ABB RAPID module: 01400AE1

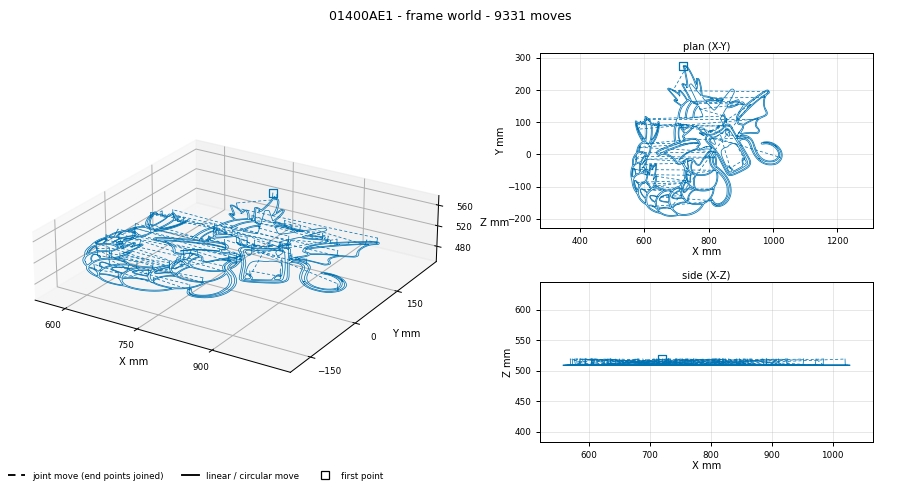
[picture p0: tool path of 01400AE1 in frame world, 9331 of 9331 moves have a stored position in this frame; points joined in program order, loops and branches not executed]
MODULE Module1
    !***********************************************************
    !
    ! Module:  Module1
    !
    ! Description:
    !   <Insert description here>
    !
    ! Author: ufabc
    !
    ! Version: 1.0
    !
    !***********************************************************


    !***********************************************************
    !
    ! Procedure main
    !
    !   This is the entry point of your program
    !
    !***********************************************************
    PROC main()
        !Add your code here
        CONST robtarget p0:=[[557.96,-192.62,509.20],[0.00299687,-0.165444,-0.986215,-0.000502744],[-1,0,0,0],[9E+09,9E+09,9E+09,9E+09,9E+09,9E+09]];

      MoveJ Offs(p0,163.0,466.8, 10), v100, z1, tool0;
MoveL Offs(p0,163.22140000000005,465.1791, 0), v100, z5, tool0;
MoveL Offs(p0,163.3808,464.47520000000003, 0), v100, z5, tool0;
MoveL Offs(p0,163.575,463.7125, 0), v100, z5, tool0;
MoveL Offs(p0,163.79919999999998,462.90479999999997, 0), v100, z5, tool0;
MoveL Offs(p0,164.0486,462.06589999999994, 0), v100, z5, tool0;
MoveL Offs(p0,164.31840000000003,461.2096, 0), v100, z5, tool0;
MoveL Offs(p0,164.6038,460.34970000000004, 0), v100, z5, tool0;
MoveL Offs(p0,164.9,459.5, 0), v100, z5, tool0;
MoveL Offs(p0,165.8568,456.4537, 0), v100, z5, tool0;
MoveL Offs(p0,166.95040000000003,452.1936000000002, 0), v100, z5, tool0;
MoveL Offs(p0,168.12560000000002,447.01789999999994, 0), v100, z5, tool0;
MoveL Offs(p0,169.3272,441.2248000000001, 0), v100, z5, tool0;
MoveL Offs(p0,170.5,435.1125, 0), v100, z5, tool0;
MoveL Offs(p0,171.5888,428.97919999999993, 0), v100, z5, tool0;
MoveL Offs(p0,172.5384,423.12309999999997, 0), v100, z5, tool0;
MoveL Offs(p0,173.29360000000003,417.8424000000001, 0), v100, z5, tool0;
MoveL Offs(p0,173.7992,413.4353, 0), v100, z5, tool0;
MoveL Offs(p0,174.0,410.2, 0), v100, z5, tool0;
MoveL Offs(p0,174.0,407.8, 0), v100, z5, tool0;
MoveL Offs(p0,169.4,410.4, 0), v100, z5, tool0;
MoveL Offs(p0,167.8938,411.19489999999996, 0), v100, z5, tool0;
MoveL Offs(p0,166.49440000000007,411.83920000000006, 0), v100, z5, tool0;
MoveL Offs(p0,165.20059999999998,412.33230000000003, 0), v100, z5, tool0;
MoveL Offs(p0,164.0112,412.67359999999996, 0), v100, z5, tool0;
MoveL Offs(p0,162.925,412.8625, 0), v100, z5, tool0;
MoveL Offs(p0,161.9408,412.8983999999999, 0), v100, z5, tool0;
MoveL Offs(p0,161.05739999999997,412.78069999999997, 0), v100, z5, tool0;
MoveL Offs(p0,160.27360000000002,412.50880000000006, 0), v100, z5, tool0;
MoveL Offs(p0,159.5882,412.08209999999997, 0), v100, z5, tool0;
MoveL Offs(p0,159.0,411.5, 0), v100, z5, tool0;
MoveL Offs(p0,158.76520000000002,411.12570000000005, 0), v100, z5, tool0;
MoveL Offs(p0,158.66960000000003,410.6416000000001, 0), v100, z5, tool0;
MoveL Offs(p0,158.72639999999998,410.01590000000004, 0), v100, z5, tool0;
MoveL Offs(p0,159.35,408.2125, 0), v100, z5, tool0;
MoveL Offs(p0,159.9432,406.9712, 0), v100, z5, tool0;
MoveL Offs(p0,160.7416,405.4611, 0), v100, z5, tool0;
MoveL Offs(p0,161.75840000000002,403.65040000000005, 0), v100, z5, tool0;
MoveL Offs(p0,163.00680000000003,401.50730000000004, 0), v100, z5, tool0;
MoveL Offs(p0,164.5,399.0, 0), v100, z5, tool0;
MoveL Offs(p0,166.88540000000003,394.95990000000006, 0), v100, z5, tool0;
MoveL Offs(p0,169.31520000000003,390.7272000000001, 0), v100, z5, tool0;
MoveL Offs(p0,171.71980000000002,386.43330000000003, 0), v100, z5, tool0;
MoveL Offs(p0,174.02960000000002,382.2096, 0), v100, z5, tool0;
MoveL Offs(p0,176.175,378.1875, 0), v100, z5, tool0;
MoveL Offs(p0,178.08639999999997,374.49839999999995, 0), v100, z5, tool0;
MoveL Offs(p0,179.6942,371.2737, 0), v100, z5, tool0;
MoveL Offs(p0,180.9288,368.64480000000003, 0), v100, z5, tool0;
MoveL Offs(p0,181.72060000000002,366.7431, 0), v100, z5, tool0;
MoveL Offs(p0,182.0,365.7, 0), v100, z5, tool0;
MoveL Offs(p0,181.59200000000004,364.89280000000014, 0), v100, z5, tool0;
MoveL Offs(p0,181.136,364.41569999999996, 0), v100, z5, tool0;
MoveL Offs(p0,180.56,363.92240000000004, 0), v100, z5, tool0;
MoveL Offs(p0,179.9,363.4375, 0), v100, z5, tool0;
MoveL Offs(p0,179.19199999999998,362.98560000000003, 0), v100, z5, tool0;
MoveL Offs(p0,178.47199999999998,362.5913, 0), v100, z5, tool0;
MoveL Offs(p0,177.776,362.27920000000006, 0), v100, z5, tool0;
MoveL Offs(p0,177.14000000000001,362.07390000000004, 0), v100, z5, tool0;
MoveL Offs(p0,176.6,362.0, 0), v100, z5, tool0;
MoveL Offs(p0,176.25680000000006,362.4672000000001, 0), v100, z5, tool0;
MoveL Offs(p0,175.8917,363.0233, 0), v100, z5, tool0;
MoveL Offs(p0,175.41440000000003,363.7696000000001, 0), v100, z5, tool0;
MoveL Offs(p0,174.8375,364.6875, 0), v100, z5, tool0;
MoveL Offs(p0,174.17360000000002,365.7584, 0), v100, z5, tool0;
MoveL Offs(p0,173.43529999999998,366.96369999999996, 0), v100, z5, tool0;
MoveL Offs(p0,172.63520000000003,368.2848, 0), v100, z5, tool0;
MoveL Offs(p0,171.7859,369.7031, 0), v100, z5, tool0;
MoveL Offs(p0,170.9,371.2, 0), v100, z5, tool0;
MoveL Offs(p0,169.93810000000002,372.75730000000004, 0), v100, z5, tool0;
MoveL Offs(p0,168.86880000000002,374.40640000000013, 0), v100, z5, tool0;
MoveL Offs(p0,167.7167,376.1131, 0), v100, z5, tool0;
MoveL Offs(p0,166.5064,377.8432, 0), v100, z5, tool0;
MoveL Offs(p0,165.2625,379.5625, 0), v100, z5, tool0;
MoveL Offs(p0,164.0096,381.23679999999996, 0), v100, z5, tool0;
MoveL Offs(p0,162.7723,382.8319, 0), v100, z5, tool0;
MoveL Offs(p0,161.57520000000002,384.31360000000006, 0), v100, z5, tool0;
MoveL Offs(p0,160.4429,385.64770000000004, 0), v100, z5, tool0;
MoveL Offs(p0,159.4,386.8, 0), v100, z5, tool0;
MoveL Offs(p0,157.8607,388.40900000000005, 0), v100, z5, tool0;
MoveL Offs(p0,156.57760000000002,389.7120000000001, 0), v100, z5, tool0;
MoveL Offs(p0,155.5129,390.733, 0), v100, z5, tool0;
MoveL Offs(p0,154.6288,391.49600000000004, 0), v100, z5, tool0;
MoveL Offs(p0,153.8875,392.025, 0), v100, z5, tool0;
MoveL Offs(p0,153.25119999999998,392.34399999999994, 0), v100, z5, tool0;
MoveL Offs(p0,152.6821,392.477, 0), v100, z5, tool0;
MoveL Offs(p0,152.1424,392.44800000000004, 0), v100, z5, tool0;
MoveL Offs(p0,151.59430000000003,392.281, 0), v100, z5, tool0;
MoveL Offs(p0,151.0,392.0, 0), v100, z5, tool0;
MoveL Offs(p0,150.4772,391.7028, 0), v100, z5, tool0;
MoveL Offs(p0,150.04560000000004,391.3984000000001, 0), v100, z5, tool0;
MoveL Offs(p0,149.70039999999997,391.06759999999997, 0), v100, z5, tool0;
MoveL Offs(p0,149.4368,390.69120000000004, 0), v100, z5, tool0;
MoveL Offs(p0,149.25,390.25, 0), v100, z5, tool0;
MoveL Offs(p0,149.13520000000003,389.7248, 0), v100, z5, tool0;
MoveL Offs(p0,149.0876,389.0964, 0), v100, z5, tool0;
MoveL Offs(p0,149.10240000000002,388.3456, 0), v100, z5, tool0;
MoveL Offs(p0,149.1748,387.45320000000004, 0), v100, z5, tool0;
MoveL Offs(p0,149.3,386.4, 0), v100, z5, tool0;
MoveL Offs(p0,149.51680000000005,384.25440000000015, 0), v100, z5, tool0;
MoveL Offs(p0,149.5502,383.5281, 0), v100, z5, tool0;
MoveL Offs(p0,149.5224,383.01120000000003, 0), v100, z5, tool0;
MoveL Offs(p0,148.98780000000002,382.5549, 0), v100, z5, tool0;
MoveL Offs(p0,148.6312,382.71360000000004, 0), v100, z5, tool0;
MoveL Offs(p0,148.1714,383.0007, 0), v100, z5, tool0;
MoveL Offs(p0,147.6,383.4, 0), v100, z5, tool0;
MoveL Offs(p0,145.2276,385.0427000000001, 0), v100, z5, tool0;
MoveL Offs(p0,142.50480000000005,386.80960000000016, 0), v100, z5, tool0;
MoveL Offs(p0,139.5432,388.6389, 0), v100, z5, tool0;
MoveL Offs(p0,136.45440000000002,390.46880000000004, 0), v100, z5, tool0;
MoveL Offs(p0,133.35,392.2375, 0), v100, z5, tool0;
MoveL Offs(p0,130.3416,393.88319999999993, 0), v100, z5, tool0;
MoveL Offs(p0,127.54079999999999,395.34409999999997, 0), v100, z5, tool0;
MoveL Offs(p0,125.0592,396.5584, 0), v100, z5, tool0;
MoveL Offs(p0,123.00840000000001,397.4643, 0), v100, z5, tool0;
MoveL Offs(p0,121.5,398.0, 0), v100, z5, tool0;
MoveL Offs(p0,120.39220000000003,398.29670000000004, 0), v100, z5, tool0;
MoveL Offs(p0,119.45360000000002,398.52560000000005, 0), v100, z5, tool0;
MoveL Offs(p0,118.6614,398.6848999999999, 0), v100, z5, tool0;
MoveL Offs(p0,117.99279999999999,398.7728000000001, 0), v100, z5, tool0;
MoveL Offs(p0,117.425,398.7875, 0), v100, z5, tool0;
MoveL Offs(p0,116.93519999999998,398.7272, 0), v100, z5, tool0;
MoveL Offs(p0,116.5006,398.5901, 0), v100, z5, tool0;
MoveL Offs(p0,116.0984,398.37440000000004, 0), v100, z5, tool0;
MoveL Offs(p0,115.3,397.7, 0), v100, z5, tool0;
MoveL Offs(p0,114.80490000000002,397.22830000000005, 0), v100, z5, tool0;
MoveL Offs(p0,114.47120000000004,396.7944000000001, 0), v100, z5, tool0;
MoveL Offs(p0,114.40630000000002,396.2501, 0), v100, z5, tool0;
MoveL Offs(p0,114.71759999999999,395.4472, 0), v100, z5, tool0;
MoveL Offs(p0,115.5125,394.2375, 0), v100, z5, tool0;
MoveL Offs(p0,116.89840000000001,392.4728, 0), v100, z5, tool0;
MoveL Offs(p0,118.9827,390.0049, 0), v100, z5, tool0;
MoveL Offs(p0,121.87280000000001,386.6856000000001, 0), v100, z5, tool0;
MoveL Offs(p0,125.67609999999999,382.36670000000004, 0), v100, z5, tool0;
MoveL Offs(p0,130.5,376.9, 0), v100, z5, tool0;
MoveL Offs(p0,141.4,364.5, 0), v100, z5, tool0;
MoveL Offs(p0,138.0,364.0, 0), v100, z5, tool0;
MoveL Offs(p0,136.66540000000003,363.7148, 0), v100, z5, tool0;
MoveL Offs(p0,135.60320000000004,363.2904000000001, 0), v100, z5, tool0;
MoveL Offs(p0,134.81580000000002,362.74359999999996, 0), v100, z5, tool0;
MoveL Offs(p0,134.3056,362.0912, 0), v100, z5, tool0;
MoveL Offs(p0,134.075,361.35, 0), v100, z5, tool0;
MoveL Offs(p0,134.1264,360.53679999999997, 0), v100, z5, tool0;
MoveL Offs(p0,134.4622,359.6684, 0), v100, z5, tool0;
MoveL Offs(p0,135.0848,358.76160000000004, 0), v100, z5, tool0;
MoveL Offs(p0,135.9966,357.83320000000003, 0), v100, z5, tool0;
MoveL Offs(p0,137.2,356.9, 0), v100, z5, tool0;
MoveL Offs(p0,137.83499999999998,356.468, 0), v100, z5, tool0;
MoveL Offs(p0,138.64400000000006,355.9040000000001, 0), v100, z5, tool0;
MoveL Offs(p0,139.603,355.226, 0), v100, z5, tool0;
MoveL Offs(p0,140.68800000000002,354.45200000000006, 0), v100, z5, tool0;
MoveL Offs(p0,141.875,353.6, 0), v100, z5, tool0;
MoveL Offs(p0,143.14000000000001,352.688, 0), v100, z5, tool0;
MoveL Offs(p0,144.459,351.73400000000004, 0), v100, z5, tool0;
MoveL Offs(p0,145.80800000000002,350.75600000000003, 0), v100, z5, tool0;
MoveL Offs(p0,147.163,349.77200000000005, 0), v100, z5, tool0;
MoveL Offs(p0,148.5,348.8, 0), v100, z5, tool0;
MoveL Offs(p0,156.6,342.9, 0), v100, z5, tool0;
MoveL Offs(p0,153.3,336.2, 0), v100, z5, tool0;
MoveL Offs(p0,152.22450000000003,333.89, 0), v100, z5, tool0;
MoveL Offs(p0,151.22400000000005,331.4240000000001, 0), v100, z5, tool0;
MoveL Offs(p0,150.30749999999998,328.838, 0), v100, z5, tool0;
MoveL Offs(p0,149.48399999999998,326.168, 0), v100, z5, tool0;
MoveL Offs(p0,148.7625,323.45, 0), v100, z5, tool0;
MoveL Offs(p0,148.152,320.72, 0), v100, z5, tool0;
MoveL Offs(p0,147.6615,318.014, 0), v100, z5, tool0;
MoveL Offs(p0,147.3,315.36800000000005, 0), v100, z5, tool0;
MoveL Offs(p0,147.07649999999998,312.81800000000004, 0), v100, z5, tool0;
MoveL Offs(p0,147.0,310.4, 0), v100, z5, tool0;
MoveL Offs(p0,146.7536,306.6048, 0), v100, z5, tool0;
MoveL Offs(p0,146.575,306.025, 0), v100, z5, tool0;
MoveL Offs(p0,146.3304,305.5472, 0), v100, z5, tool0;
MoveL Offs(p0,146.0102,305.1486, 0), v100, z5, tool0;
MoveL Offs(p0,145.6048,304.80640000000005, 0), v100, z5, tool0;
MoveL Offs(p0,145.1046,304.4978, 0), v100, z5, tool0;
MoveL Offs(p0,144.5,304.2, 0), v100, z5, tool0;
MoveL Offs(p0,143.69200000000004,303.78720000000004, 0), v100, z5, tool0;
MoveL Offs(p0,143.321,303.54929999999996, 0), v100, z5, tool0;
MoveL Offs(p0,142.98000000000002,303.2976, 0), v100, z5, tool0;
MoveL Offs(p0,142.675,303.0375, 0), v100, z5, tool0;
MoveL Offs(p0,142.412,302.7744, 0), v100, z5, tool0;
MoveL Offs(p0,142.197,302.5137, 0), v100, z5, tool0;
MoveL Offs(p0,142.036,302.2608, 0), v100, z5, tool0;
MoveL Offs(p0,141.935,302.02110000000005, 0), v100, z5, tool0;
MoveL Offs(p0,141.9,301.8, 0), v100, z5, tool0;
MoveL Offs(p0,141.7,299.85, 0), v100, z5, tool0;
MoveL Offs(p0,141.65519999999998,299.3088, 0), v100, z5, tool0;
MoveL Offs(p0,141.6116,298.7424, 0), v100, z5, tool0;
MoveL Offs(p0,141.5704,298.1616, 0), v100, z5, tool0;
MoveL Offs(p0,141.5328,297.5772, 0), v100, z5, tool0;
MoveL Offs(p0,141.5,297.0, 0), v100, z5, tool0;
MoveL Offs(p0,141.22160000000002,295.45040000000006, 0), v100, z5, tool0;
MoveL Offs(p0,140.9744,294.4071, 0), v100, z5, tool0;
MoveL Offs(p0,140.6648,293.2192, 0), v100, z5, tool0;
MoveL Offs(p0,140.3,291.9125, 0), v100, z5, tool0;
MoveL Offs(p0,139.88719999999998,290.51279999999997, 0), v100, z5, tool0;
MoveL Offs(p0,139.4336,289.04589999999996, 0), v100, z5, tool0;
MoveL Offs(p0,138.94639999999998,287.5376, 0), v100, z5, tool0;
MoveL Offs(p0,138.4328,286.0137, 0), v100, z5, tool0;
MoveL Offs(p0,137.9,284.5, 0), v100, z5, tool0;
MoveL Offs(p0,137.07820000000004,282.18640000000005, 0), v100, z5, tool0;
MoveL Offs(p0,136.40160000000006,280.1512000000001, 0), v100, z5, tool0;
MoveL Offs(p0,135.8534,278.28279999999995, 0), v100, z5, tool0;
MoveL Offs(p0,135.41680000000002,276.4696, 0), v100, z5, tool0;
MoveL Offs(p0,135.075,274.6, 0), v100, z5, tool0;
MoveL Offs(p0,134.81119999999999,272.56239999999997, 0), v100, z5, tool0;
MoveL Offs(p0,134.6086,270.2452, 0), v100, z5, tool0;
MoveL Offs(p0,134.4504,267.53679999999997, 0), v100, z5, tool0;
MoveL Offs(p0,134.31980000000001,264.3256, 0), v100, z5, tool0;
MoveL Offs(p0,134.2,260.5, 0), v100, z5, tool0;
MoveL Offs(p0,134.6125,243.425, 0), v100, z5, tool0;
MoveL Offs(p0,134.97039999999998,240.6424, 0), v100, z5, tool0;
MoveL Offs(p0,135.4327,237.92219999999998, 0), v100, z5, tool0;
MoveL Offs(p0,136.00480000000002,235.2008, 0), v100, z5, tool0;
MoveL Offs(p0,136.6921,232.4146, 0), v100, z5, tool0;
MoveL Offs(p0,137.5,229.5, 0), v100, z5, tool0;
MoveL Offs(p0,137.15169999999998,227.925, 0), v100, z5, tool0;
MoveL Offs(p0,136.46640000000002,227.36399999999998, 0), v100, z5, tool0;
MoveL Offs(p0,135.3875,226.725, 0), v100, z5, tool0;
MoveL Offs(p0,133.8496,225.97200000000004, 0), v100, z5, tool0;
MoveL Offs(p0,131.78730000000002,225.06900000000002, 0), v100, z5, tool0;
MoveL Offs(p0,129.1352,223.98000000000002, 0), v100, z5, tool0;
MoveL Offs(p0,125.8279,222.669, 0), v100, z5, tool0;
MoveL Offs(p0,121.8,221.1, 0), v100, z5, tool0;
MoveL Offs(p0,115.05690000000001,218.44700000000003, 0), v100, z5, tool0;
MoveL Offs(p0,108.97920000000002,216.00400000000008, 0), v100, z5, tool0;
MoveL Offs(p0,103.55429999999998,213.76500000000001, 0), v100, z5, tool0;
MoveL Offs(p0,98.7696,211.72400000000002, 0), v100, z5, tool0;
MoveL Offs(p0,94.6125,209.875, 0), v100, z5, tool0;
MoveL Offs(p0,91.07039999999999,208.212, 0), v100, z5, tool0;
MoveL Offs(p0,88.1307,206.72899999999998, 0), v100, z5, tool0;
MoveL Offs(p0,85.7808,205.42, 0), v100, z5, tool0;
MoveL Offs(p0,84.0081,204.279, 0), v100, z5, tool0;
MoveL Offs(p0,82.8,203.3, 0), v100, z5, tool0;
MoveL Offs(p0,81.75000000000001,202.14080000000004, 0), v100, z5, tool0;
MoveL Offs(p0,80.94000000000003,200.95040000000006, 0), v100, z5, tool0;
MoveL Offs(p0,80.37,199.73959999999997, 0), v100, z5, tool0;
MoveL Offs(p0,80.04,198.5192, 0), v100, z5, tool0;
MoveL Offs(p0,79.95,197.3, 0), v100, z5, tool0;
MoveL Offs(p0,80.1,196.09279999999998, 0), v100, z5, tool0;
MoveL Offs(p0,80.49000000000001,194.90839999999997, 0), v100, z5, tool0;
MoveL Offs(p0,81.12,193.7576, 0), v100, z5, tool0;
MoveL Offs(p0,81.99000000000001,192.65120000000002, 0), v100, z5, tool0;
MoveL Offs(p0,83.1,191.6, 0), v100, z5, tool0;
MoveL Offs(p0,84.1761,190.75700000000003, 0), v100, z5, tool0;
MoveL Offs(p0,85.19280000000003,190.08800000000002, 0), v100, z5, tool0;
MoveL Offs(p0,86.1627,189.59300000000002, 0), v100, z5, tool0;
MoveL Offs(p0,87.0984,189.272, 0), v100, z5, tool0;
MoveL Offs(p0,88.0125,189.125, 0), v100, z5, tool0;
MoveL Offs(p0,88.91760000000001,189.152, 0), v100, z5, tool0;
MoveL Offs(p0,89.82629999999999,189.353, 0), v100, z5, tool0;
MoveL Offs(p0,90.75120000000001,189.728, 0), v100, z5, tool0;
MoveL Offs(p0,91.70490000000001,190.277, 0), v100, z5, tool0;
MoveL Offs(p0,92.7,191.0, 0), v100, z5, tool0;
MoveL Offs(p0,94.55320000000002,192.03410000000002, 0), v100, z5, tool0;
MoveL Offs(p0,96.88160000000002,192.68480000000002, 0), v100, z5, tool0;
MoveL Offs(p0,99.60839999999999,192.9647, 0), v100, z5, tool0;
MoveL Offs(p0,102.65680000000002,192.88640000000004, 0), v100, z5, tool0;
MoveL Offs(p0,105.95,192.4625, 0), v100, z5, tool0;
MoveL Offs(p0,109.41120000000001,191.7056, 0), v100, z5, tool0;
MoveL Offs(p0,112.9636,190.6283, 0), v100, z5, tool0;
MoveL Offs(p0,116.53040000000001,189.24320000000003, 0), v100, z5, tool0;
MoveL Offs(p0,120.03479999999999,187.56289999999998, 0), v100, z5, tool0;
MoveL Offs(p0,123.4,185.6, 0), v100, z5, tool0;
MoveL Offs(p0,125.15720000000002,184.40070000000003, 0), v100, z5, tool0;
MoveL Offs(p0,126.88560000000003,183.08560000000006, 0), v100, z5, tool0;
MoveL Offs(p0,128.5804,181.65890000000002, 0), v100, z5, tool0;
MoveL Offs(p0,130.23680000000002,180.1248, 0), v100, z5, tool0;
MoveL Offs(p0,131.85,178.4875, 0), v100, z5, tool0;
MoveL Offs(p0,133.4152,176.75119999999998, 0), v100, z5, tool0;
MoveL Offs(p0,134.92759999999998,174.9201, 0), v100, z5, tool0;
MoveL Offs(p0,136.38240000000002,172.9984, 0), v100, z5, tool0;
MoveL Offs(p0,137.7748,170.99030000000002, 0), v100, z5, tool0;
MoveL Offs(p0,139.1,168.9, 0), v100, z5, tool0;
MoveL Offs(p0,140.6022,166.75030000000004, 0), v100, z5, tool0;
MoveL Offs(p0,142.2136,164.92640000000003, 0), v100, z5, tool0;
MoveL Offs(p0,143.91140000000001,163.4361, 0), v100, z5, tool0;
MoveL Offs(p0,145.6728,162.2872, 0), v100, z5, tool0;
MoveL Offs(p0,147.475,161.4875, 0), v100, z5, tool0;
MoveL Offs(p0,149.2952,161.04479999999998, 0), v100, z5, tool0;
MoveL Offs(p0,151.1106,160.96689999999998, 0), v100, z5, tool0;
MoveL Offs(p0,152.8984,161.2616, 0), v100, z5, tool0;
MoveL Offs(p0,154.63580000000002,161.93670000000003, 0), v100, z5, tool0;
MoveL Offs(p0,156.3,163.0, 0), v100, z5, tool0;
MoveL Offs(p0,158.9,165.1, 0), v100, z5, tool0;
MoveL Offs(p0,161.4,160.3, 0), v100, z5, tool0;
MoveL Offs(p0,161.84230000000002,159.48710000000003, 0), v100, z5, tool0;
MoveL Offs(p0,162.32240000000007,158.6208000000001, 0), v100, z5, tool0;
MoveL Offs(p0,162.83009999999996,157.7197, 0), v100, z5, tool0;
MoveL Offs(p0,163.35520000000002,156.8024, 0), v100, z5, tool0;
MoveL Offs(p0,163.8875,155.8875, 0), v100, z5, tool0;
MoveL Offs(p0,164.41680000000002,154.9936, 0), v100, z5, tool0;
MoveL Offs(p0,164.9329,154.1393, 0), v100, z5, tool0;
MoveL Offs(p0,165.42560000000003,153.34320000000002, 0), v100, z5, tool0;
MoveL Offs(p0,165.8847,152.6239, 0), v100, z5, tool0;
MoveL Offs(p0,166.3,152.0, 0), v100, z5, tool0;
MoveL Offs(p0,166.89770000000001,151.1158, 0), v100, z5, tool0;
MoveL Offs(p0,167.37360000000007,150.36240000000004, 0), v100, z5, tool0;
MoveL Offs(p0,167.7319,149.7086, 0), v100, z5, tool0;
MoveL Offs(p0,167.97680000000003,149.1232, 0), v100, z5, tool0;
MoveL Offs(p0,168.1125,148.575, 0), v100, z5, tool0;
MoveL Offs(p0,168.1432,148.0328, 0), v100, z5, tool0;
MoveL Offs(p0,168.0731,147.4654, 0), v100, z5, tool0;
MoveL Offs(p0,167.90640000000002,146.84160000000003, 0), v100, z5, tool0;
MoveL Offs(p0,167.6473,146.1302, 0), v100, z5, tool0;
MoveL Offs(p0,167.3,145.3, 0), v100, z5, tool0;
MoveL Offs(p0,166.69410000000002,143.6099, 0), v100, z5, tool0;
MoveL Offs(p0,166.19680000000005,141.73920000000004, 0), v100, z5, tool0;
MoveL Offs(p0,165.8087,139.7173, 0), v100, z5, tool0;
MoveL Offs(p0,165.5304,137.5736, 0), v100, z5, tool0;
MoveL Offs(p0,165.3625,135.3375, 0), v100, z5, tool0;
MoveL Offs(p0,165.3056,133.0384, 0), v100, z5, tool0;
MoveL Offs(p0,165.3603,130.7057, 0), v100, z5, tool0;
MoveL Offs(p0,165.5272,128.36880000000002, 0), v100, z5, tool0;
MoveL Offs(p0,165.8069,126.05709999999999, 0), v100, z5, tool0;
MoveL Offs(p0,166.2,123.8, 0), v100, z5, tool0;
MoveL Offs(p0,167.6,117.1, 0), v100, z5, tool0;
MoveL Offs(p0,163.8,113.3, 0), v100, z5, tool0;
MoveL Offs(p0,162.6265,112.02490000000003, 0), v100, z5, tool0;
MoveL Offs(p0,161.36000000000007,110.41920000000002, 0), v100, z5, tool0;
MoveL Offs(p0,160.05149999999998,108.5723, 0), v100, z5, tool0;
MoveL Offs(p0,158.752,106.57360000000001, 0), v100, z5, tool0;
MoveL Offs(p0,157.5125,104.5125, 0), v100, z5, tool0;
MoveL Offs(p0,156.384,102.47840000000001, 0), v100, z5, tool0;
MoveL Offs(p0,155.41750000000002,100.5607, 0), v100, z5, tool0;
MoveL Offs(p0,154.66400000000002,98.84880000000001, 0), v100, z5, tool0;
MoveL Offs(p0,154.1745,97.4321, 0), v100, z5, tool0;
MoveL Offs(p0,154.0,96.4, 0), v100, z5, tool0;
MoveL Offs(p0,153.78480000000002,95.93920000000003, 0), v100, z5, tool0;
MoveL Offs(p0,153.53019999999998,95.68629999999999, 0), v100, z5, tool0;
MoveL Offs(p0,153.1904,95.4256, 0), v100, z5, tool0;
MoveL Offs(p0,152.775,95.1625, 0), v100, z5, tool0;
MoveL Offs(p0,152.2936,94.9024, 0), v100, z5, tool0;
MoveL Offs(p0,151.7558,94.6507, 0), v100, z5, tool0;
MoveL Offs(p0,151.1712,94.4128, 0), v100, z5, tool0;
MoveL Offs(p0,150.54940000000002,94.1941, 0), v100, z5, tool0;
MoveL Offs(p0,149.9,94.0, 0), v100, z5, tool0;
MoveL Offs(p0,147.96450000000004,93.4209, 0), v100, z5, tool0;
MoveL Offs(p0,145.96,92.71520000000002, 0), v100, z5, tool0;
MoveL Offs(p0,143.91950000000003,91.9003, 0), v100, z5, tool0;
MoveL Offs(p0,141.876,90.99360000000001, 0), v100, z5, tool0;
MoveL Offs(p0,139.8625,90.0125, 0), v100, z5, tool0;
MoveL Offs(p0,137.91199999999998,88.9744, 0), v100, z5, tool0;
MoveL Offs(p0,136.05749999999998,87.89669999999998, 0), v100, z5, tool0;
MoveL Offs(p0,134.33200000000002,86.7968, 0), v100, z5, tool0;
MoveL Offs(p0,132.76850000000002,85.69210000000001, 0), v100, z5, tool0;
MoveL Offs(p0,131.4,84.6, 0), v100, z5, tool0;
MoveL Offs(p0,130.41080000000002,83.758, 0), v100, z5, tool0;
MoveL Offs(p0,129.57040000000006,83.08400000000002, 0), v100, z5, tool0;
MoveL Offs(p0,128.82959999999997,82.566, 0), v100, z5, tool0;
MoveL Offs(p0,128.13920000000002,82.19200000000001, 0), v100, z5, tool0;
MoveL Offs(p0,127.45,81.95, 0), v100, z5, tool0;
MoveL Offs(p0,126.71279999999999,81.828, 0), v100, z5, tool0;
MoveL Offs(p0,125.87839999999998,81.814, 0), v100, z5, tool0;
MoveL Offs(p0,124.89760000000001,81.896, 0), v100, z5, tool0;
MoveL Offs(p0,123.7212,82.06200000000001, 0), v100, z5, tool0;
MoveL Offs(p0,122.3,82.3, 0), v100, z5, tool0;
MoveL Offs(p0,120.27520000000007,82.54000000000002, 0), v100, z5, tool0;
MoveL Offs(p0,119.20129999999999,82.61499999999998, 0), v100, z5, tool0;
MoveL Offs(p0,118.1016,82.66, 0), v100, z5, tool0;
MoveL Offs(p0,116.9875,82.675, 0), v100, z5, tool0;
MoveL Offs(p0,115.87039999999999,82.66, 0), v100, z5, tool0;
MoveL Offs(p0,114.76169999999999,82.61499999999998, 0), v100, z5, tool0;
MoveL Offs(p0,113.67280000000001,82.54, 0), v100, z5, tool0;
MoveL Offs(p0,110.27420000000004,82.06380000000001, 0), v100, z5, tool0;
MoveL Offs(p0,109.15360000000003,81.89840000000002, 0), v100, z5, tool0;
MoveL Offs(p0,108.20340000000002,81.8086, 0), v100, z5, tool0;
MoveL Offs(p0,107.38879999999999,81.7992, 0), v100, z5, tool0;
MoveL Offs(p0,106.675,81.875, 0), v100, z5, tool0;
MoveL Offs(p0,106.0272,82.04080000000002, 0), v100, z5, tool0;
MoveL Offs(p0,104.7904,82.66159999999999, 0), v100, z5, tool0;
MoveL Offs(p0,104.1318,83.12620000000001, 0), v100, z5, tool0;
MoveL Offs(p0,103.4,83.7, 0), v100, z5, tool0;
MoveL Offs(p0,102.407,84.41580000000002, 0), v100, z5, tool0;
MoveL Offs(p0,101.24000000000002,85.11840000000002, 0), v100, z5, tool0;
MoveL Offs(p0,99.917,85.8006, 0), v100, z5, tool0;
MoveL Offs(p0,98.456,86.4552, 0), v100, z5, tool0;
MoveL Offs(p0,96.875,87.075, 0), v100, z5, tool0;
MoveL Offs(p0,95.19200000000001,87.6528, 0), v100, z5, tool0;
MoveL Offs(p0,93.425,88.1814, 0), v100, z5, tool0;
MoveL Offs(p0,91.59200000000001,88.65360000000001, 0), v100, z5, tool0;
MoveL Offs(p0,89.71100000000001,89.0622, 0), v100, z5, tool0;
MoveL Offs(p0,87.8,89.4, 0), v100, z5, tool0;
MoveL Offs(p0,86.20480000000002,89.77600000000002, 0), v100, z5, tool0;
MoveL Offs(p0,85.5347,90.039, 0), v100, z5, tool0;
MoveL Offs(p0,84.92640000000002,90.36800000000001, 0), v100, z5, tool0;
MoveL Offs(p0,84.3625,90.775, 0), v100, z5, tool0;
MoveL Offs(p0,83.8256,91.27199999999999, 0), v100, z5, tool0;
MoveL Offs(p0,83.2983,91.87100000000001, 0), v100, z5, tool0;
MoveL Offs(p0,82.76320000000001,92.584, 0), v100, z5, tool0;
MoveL Offs(p0,82.2029,93.423, 0), v100, z5, tool0;
MoveL Offs(p0,81.6,94.4, 0), v100, z5, tool0;
MoveL Offs(p0,81.1722,95.0939, 0), v100, z5, tool0;
MoveL Offs(p0,80.73360000000002,95.78720000000001, 0), v100, z5, tool0;
MoveL Offs(p0,80.2914,96.4673, 0), v100, z5, tool0;
MoveL Offs(p0,79.8528,97.12160000000002, 0), v100, z5, tool0;
MoveL Offs(p0,79.425,97.7375, 0), v100, z5, tool0;
MoveL Offs(p0,79.01520000000001,98.3024, 0), v100, z5, tool0;
MoveL Offs(p0,78.6306,98.80369999999999, 0), v100, z5, tool0;
MoveL Offs(p0,78.2784,99.2288, 0), v100, z5, tool0;
MoveL Offs(p0,77.96580000000002,99.5651, 0), v100, z5, tool0;
MoveL Offs(p0,77.7,99.8, 0), v100, z5, tool0;
MoveL Offs(p0,77.38240000000002,100.11720000000001, 0), v100, z5, tool0;
MoveL Offs(p0,77.15120000000003,100.48960000000002, 0), v100, z5, tool0;
MoveL Offs(p0,77.0088,100.94839999999999, 0), v100, z5, tool0;
MoveL Offs(p0,76.95760000000001,101.52480000000001, 0), v100, z5, tool0;
MoveL Offs(p0,77.0,102.25, 0), v100, z5, tool0;
MoveL Offs(p0,77.13839999999999,103.1552, 0), v100, z5, tool0;
MoveL Offs(p0,77.37519999999999,104.27159999999999, 0), v100, z5, tool0;
MoveL Offs(p0,78.15360000000001,107.26280000000001, 0), v100, z5, tool0;
MoveL Offs(p0,78.7,109.2, 0), v100, z5, tool0;
MoveL Offs(p0,79.4558,112.0721, 0), v100, z5, tool0;
MoveL Offs(p0,80.04240000000001,114.74080000000004, 0), v100, z5, tool0;
MoveL Offs(p0,80.45860000000002,117.19469999999998, 0), v100, z5, tool0;
MoveL Offs(p0,80.70320000000001,119.42240000000001, 0), v100, z5, tool0;
MoveL Offs(p0,80.775,121.4125, 0), v100, z5, tool0;
MoveL Offs(p0,80.6728,123.15360000000001, 0), v100, z5, tool0;
MoveL Offs(p0,80.3954,124.63429999999998, 0), v100, z5, tool0;
MoveL Offs(p0,79.9416,125.84320000000002, 0), v100, z5, tool0;
MoveL Offs(p0,79.31020000000001,126.7689, 0), v100, z5, tool0;
MoveL Offs(p0,78.5,127.4, 0), v100, z5, tool0;
MoveL Offs(p0,77.85840000000003,127.74480000000003, 0), v100, z5, tool0;
MoveL Offs(p0,77.55859999999998,127.9022, 0), v100, z5, tool0;
MoveL Offs(p0,77.2792,128.0464, 0), v100, z5, tool0;
MoveL Offs(p0,77.025,128.175, 0), v100, z5, tool0;
MoveL Offs(p0,76.80080000000001,128.2856, 0), v100, z5, tool0;
MoveL Offs(p0,76.6114,128.3758, 0), v100, z5, tool0;
MoveL Offs(p0,76.46160000000002,128.44320000000002, 0), v100, z5, tool0;
MoveL Offs(p0,76.35620000000002,128.4854, 0), v100, z5, tool0;
MoveL Offs(p0,76.3,128.5, 0), v100, z5, tool0;
MoveL Offs(p0,76.57359999999998,130.5736, 0), v100, z5, tool0;
MoveL Offs(p0,76.6878,131.22930000000002, 0), v100, z5, tool0;
MoveL Offs(p0,76.8152,131.94320000000002, 0), v100, z5, tool0;
MoveL Offs(p0,76.95340000000002,132.7039, 0), v100, z5, tool0;
MoveL Offs(p0,77.1,133.5, 0), v100, z5, tool0;
MoveL Offs(p0,77.50320000000002,135.68640000000002, 0), v100, z5, tool0;
MoveL Offs(p0,77.73179999999999,137.10809999999998, 0), v100, z5, tool0;
MoveL Offs(p0,77.9736,138.70319999999998, 0), v100, z5, tool0;
MoveL Offs(p0,78.225,140.4375, 0), v100, z5, tool0;
MoveL Offs(p0,78.48239999999998,142.2768, 0), v100, z5, tool0;
MoveL Offs(p0,78.7422,144.1869, 0), v100, z5, tool0;
MoveL Offs(p0,79.0008,146.13360000000003, 0), v100, z5, tool0;
MoveL Offs(p0,79.25460000000001,148.08270000000002, 0), v100, z5, tool0;
MoveL Offs(p0,79.5,150.0, 0), v100, z5, tool0;
MoveL Offs(p0,79.8237,152.85370000000006, 0), v100, z5, tool0;
MoveL Offs(p0,80.07360000000001,155.21360000000004, 0), v100, z5, tool0;
MoveL Offs(p0,80.24789999999999,157.1379, 0), v100, z5, tool0;
MoveL Offs(p0,80.3448,158.68480000000002, 0), v100, z5, tool0;
MoveL Offs(p0,80.3625,159.9125, 0), v100, z5, tool0;
MoveL Offs(p0,80.29920000000001,160.8792, 0), v100, z5, tool0;
MoveL Offs(p0,80.1531,161.6431, 0), v100, z5, tool0;
MoveL Offs(p0,79.92240000000001,162.2624, 0), v100, z5, tool0;
MoveL Offs(p0,79.2,163.3, 0), v100, z5, tool0;
MoveL Offs(p0,78.3468,164.1183, 0), v100, z5, tool0;
MoveL Offs(p0,77.5224,164.65040000000005, 0), v100, z5, tool0;
MoveL Offs(p0,76.71959999999999,164.8921, 0), v100, z5, tool0;
MoveL Offs(p0,75.9312,164.8392, 0), v100, z5, tool0;
MoveL Offs(p0,75.15,164.4875, 0), v100, z5, tool0;
MoveL Offs(p0,74.3688,163.8328, 0), v100, z5, tool0;
MoveL Offs(p0,73.5804,162.8709, 0), v100, z5, tool0;
MoveL Offs(p0,72.7776,161.5976, 0), v100, z5, tool0;
MoveL Offs(p0,71.95320000000001,160.0087, 0), v100, z5, tool0;
MoveL Offs(p0,71.1,158.1, 0), v100, z5, tool0;
MoveL Offs(p0,68.5,151.7, 0), v100, z5, tool0;
MoveL Offs(p0,66.0,157.3, 0), v100, z5, tool0;
MoveL Offs(p0,65.60230000000001,158.21290000000002, 0), v100, z5, tool0;
MoveL Offs(p0,65.19440000000002,159.08320000000003, 0), v100, z5, tool0;
MoveL Offs(p0,64.7841,159.8983, 0), v100, z5, tool0;
MoveL Offs(p0,64.3792,160.6456, 0), v100, z5, tool0;
MoveL Offs(p0,63.9875,161.3125, 0), v100, z5, tool0;
MoveL Offs(p0,63.61679999999999,161.88639999999998, 0), v100, z5, tool0;
MoveL Offs(p0,63.2749,162.3547, 0), v100, z5, tool0;
MoveL Offs(p0,62.9696,162.7048, 0), v100, z5, tool0;
MoveL Offs(p0,62.7087,162.9241, 0), v100, z5, tool0;
MoveL Offs(p0,62.5,163.0, 0), v100, z5, tool0;
MoveL Offs(p0,61.046400000000006,162.70640000000003, 0), v100, z5, tool0;
MoveL Offs(p0,60.442600000000006,162.3781, 0), v100, z5, tool0;
MoveL Offs(p0,59.919200000000004,161.9232, 0), v100, z5, tool0;
MoveL Offs(p0,59.475,161.3375, 0), v100, z5, tool0;
MoveL Offs(p0,59.108799999999995,160.61679999999998, 0), v100, z5, tool0;
MoveL Offs(p0,58.819399999999995,159.7569, 0), v100, z5, tool0;
MoveL Offs(p0,58.6056,158.7536, 0), v100, z5, tool0;
MoveL Offs(p0,58.4662,157.6027, 0), v100, z5, tool0;
MoveL Offs(p0,58.4,156.3, 0), v100, z5, tool0;
MoveL Offs(p0,58.113600000000005,146.1064, 0), v100, z5, tool0;
MoveL Offs(p0,58.0,144.275, 0), v100, z5, tool0;
MoveL Offs(p0,57.8744,142.7856, 0), v100, z5, tool0;
MoveL Offs(p0,57.739200000000004,141.66580000000002, 0), v100, z5, tool0;
MoveL Offs(p0,57.59680000000001,140.94320000000002, 0), v100, z5, tool0;
MoveL Offs(p0,57.4496,140.64540000000002, 0), v100, z5, tool0;
MoveL Offs(p0,57.3,140.8, 0), v100, z5, tool0;
MoveL Offs(p0,57.0172,141.25320000000005, 0), v100, z5, tool0;
MoveL Offs(p0,56.609600000000015,141.59360000000004, 0), v100, z5, tool0;
MoveL Offs(p0,56.108399999999996,141.82240000000002, 0), v100, z5, tool0;
MoveL Offs(p0,55.54480000000001,141.94080000000002, 0), v100, z5, tool0;
MoveL Offs(p0,54.95,141.95, 0), v100, z5, tool0;
MoveL Offs(p0,54.3552,141.8512, 0), v100, z5, tool0;
MoveL Offs(p0,53.791599999999995,141.6456, 0), v100, z5, tool0;
MoveL Offs(p0,53.2904,141.33440000000002, 0), v100, z5, tool0;
MoveL Offs(p0,52.6,140.4, 0), v100, z5, tool0;
MoveL Offs(p0,52.3381,139.3605, 0), v100, z5, tool0;
MoveL Offs(p0,52.2592,138.936, 0), v100, z5, tool0;
MoveL Offs(p0,52.1875,138.4875, 0), v100, z5, tool0;
MoveL Offs(p0,52.12480000000001,138.02399999999997, 0), v100, z5, tool0;
MoveL Offs(p0,52.07289999999999,137.55450000000002, 0), v100, z5, tool0;
MoveL Offs(p0,52.0336,137.08800000000002, 0), v100, z5, tool0;
MoveL Offs(p0,52.0087,136.6335, 0), v100, z5, tool0;
MoveL Offs(p0,52.0,136.2, 0), v100, z5, tool0;
MoveL Offs(p0,51.75,133.95, 0), v100, z5, tool0;
MoveL Offs(p0,51.654399999999995,133.54319999999998, 0), v100, z5, tool0;
MoveL Offs(p0,51.5492,133.1676, 0), v100, z5, tool0;
MoveL Offs(p0,51.436800000000005,132.8304, 0), v100, z5, tool0;
MoveL Offs(p0,51.3196,132.53879999999998, 0), v100, z5, tool0;
MoveL Offs(p0,51.2,132.3, 0), v100, z5, tool0;
MoveL Offs(p0,50.869699999999995,132.76709999999997, 0), v100, z5, tool0;
MoveL Offs(p0,50.77440000000001,133.3272, 0), v100, z5, tool0;
MoveL Offs(p0,50.6875,134.0625, 0), v100, z5, tool0;
MoveL Offs(p0,50.6096,134.9568, 0), v100, z5, tool0;
MoveL Offs(p0,50.5413,135.9939, 0), v100, z5, tool0;
MoveL Offs(p0,50.483200000000004,137.1576, 0), v100, z5, tool0;
MoveL Offs(p0,50.435900000000004,138.4317, 0), v100, z5, tool0;
MoveL Offs(p0,50.4,139.8, 0), v100, z5, tool0;
MoveL Offs(p0,50.10560000000001,146.1312, 0), v100, z5, tool0;
MoveL Offs(p0,49.9375,147.4875, 0), v100, z5, tool0;
MoveL Offs(p0,49.730399999999996,148.7568, 0), v100, z5, tool0;
MoveL Offs(p0,49.4837,149.9409, 0), v100, z5, tool0;
MoveL Offs(p0,49.1968,151.04160000000002, 0), v100, z5, tool0;
MoveL Offs(p0,48.8691,152.0607, 0), v100, z5, tool0;
MoveL Offs(p0,48.5,153.0, 0), v100, z5, tool0;
MoveL Offs(p0,47.906000000000006,154.59890000000001, 0), v100, z5, tool0;
MoveL Offs(p0,47.44400000000001,156.05920000000003, 0), v100, z5, tool0;
MoveL Offs(p0,47.114,157.41629999999998, 0), v100, z5, tool0;
MoveL Offs(p0,46.916000000000004,158.70560000000003, 0), v100, z5, tool0;
MoveL Offs(p0,46.85,159.9625, 0), v100, z5, tool0;
MoveL Offs(p0,46.916000000000004,161.22240000000002, 0), v100, z5, tool0;
MoveL Offs(p0,47.114,162.5207, 0), v100, z5, tool0;
MoveL Offs(p0,47.444,163.89280000000002, 0), v100, z5, tool0;
MoveL Offs(p0,47.906000000000006,165.3741, 0), v100, z5, tool0;
MoveL Offs(p0,48.77490000000001,167.8154, 0), v100, z5, tool0;
MoveL Offs(p0,49.055200000000006,168.74720000000005, 0), v100, z5, tool0;
MoveL Offs(p0,49.3343,169.7738, 0), v100, z5, tool0;
MoveL Offs(p0,49.6056,170.87359999999998, 0), v100, z5, tool0;
MoveL Offs(p0,49.8625,172.025, 0), v100, z5, tool0;
MoveL Offs(p0,50.098400000000005,173.20639999999997, 0), v100, z5, tool0;
MoveL Offs(p0,50.3067,174.3962, 0), v100, z5, tool0;
MoveL Offs(p0,50.4808,175.5728, 0), v100, z5, tool0;
MoveL Offs(p0,50.61410000000001,176.71460000000002, 0), v100, z5, tool0;
MoveL Offs(p0,50.7,177.8, 0), v100, z5, tool0;
MoveL Offs(p0,51.02880000000001,180.55600000000007, 0), v100, z5, tool0;
MoveL Offs(p0,51.2337,181.66549999999998, 0), v100, z5, tool0;
MoveL Offs(p0,51.482400000000005,182.64000000000001, 0), v100, z5, tool0;
MoveL Offs(p0,51.7875,183.5125, 0), v100, z5, tool0;
MoveL Offs(p0,52.1616,184.316, 0), v100, z5, tool0;
MoveL Offs(p0,52.6173,185.08350000000002, 0), v100, z5, tool0;
MoveL Offs(p0,53.1672,185.848, 0), v100, z5, tool0;
MoveL Offs(p0,53.8239,186.6425, 0), v100, z5, tool0;
MoveL Offs(p0,54.6,187.5, 0), v100, z5, tool0;
MoveL Offs(p0,56.03090000000001,189.19780000000003, 0), v100, z5, tool0;
MoveL Offs(p0,57.32320000000002,191.05040000000002, 0), v100, z5, tool0;
MoveL Offs(p0,58.4763,193.05659999999997, 0), v100, z5, tool0;
MoveL Offs(p0,59.48960000000001,195.2152, 0), v100, z5, tool0;
MoveL Offs(p0,60.3625,197.525, 0), v100, z5, tool0;
MoveL Offs(p0,61.09439999999999,199.9848, 0), v100, z5, tool0;
MoveL Offs(p0,61.6847,202.59339999999997, 0), v100, z5, tool0;
MoveL Offs(p0,62.132799999999996,205.3496, 0), v100, z5, tool0;
MoveL Offs(p0,62.438100000000006,208.2522, 0), v100, z5, tool0;
MoveL Offs(p0,62.6,211.3, 0), v100, z5, tool0;
MoveL Offs(p0,62.8583,216.4858, 0), v100, z5, tool0;
MoveL Offs(p0,62.9936,217.74960000000002, 0), v100, z5, tool0;
MoveL Offs(p0,63.1625,218.825, 0), v100, z5, tool0;
MoveL Offs(p0,63.3704,219.7384, 0), v100, z5, tool0;
MoveL Offs(p0,63.622699999999995,220.51619999999997, 0), v100, z5, tool0;
MoveL Offs(p0,63.924800000000005,221.1848, 0), v100, z5, tool0;
MoveL Offs(p0,64.2821,221.7706, 0), v100, z5, tool0;
MoveL Offs(p0,64.7,222.3, 0), v100, z5, tool0;
MoveL Offs(p0,66.21270000000001,224.07080000000002, 0), v100, z5, tool0;
MoveL Offs(p0,67.78960000000002,226.05040000000002, 0), v100, z5, tool0;
MoveL Offs(p0,69.3989,228.18959999999998, 0), v100, z5, tool0;
MoveL Offs(p0,71.0088,230.43920000000003, 0), v100, z5, tool0;
MoveL Offs(p0,72.5875,232.75, 0), v100, z5, tool0;
MoveL Offs(p0,74.1032,235.0728, 0), v100, z5, tool0;
MoveL Offs(p0,75.5241,237.3584, 0), v100, z5, tool0;
MoveL Offs(p0,76.8184,239.5576, 0), v100, z5, tool0;
MoveL Offs(p0,77.9543,241.6212, 0), v100, z5, tool0;
MoveL Offs(p0,78.9,243.5, 0), v100, z5, tool0;
MoveL Offs(p0,80.70000000000002,247.60530000000003, 0), v100, z5, tool0;
MoveL Offs(p0,82.36800000000002,252.00640000000004, 0), v100, z5, tool0;
MoveL Offs(p0,83.886,256.6211, 0), v100, z5, tool0;
MoveL Offs(p0,85.236,261.3672, 0), v100, z5, tool0;
MoveL Offs(p0,86.4,266.1625, 0), v100, z5, tool0;
MoveL Offs(p0,87.36,270.9248, 0), v100, z5, tool0;
MoveL Offs(p0,88.098,275.5719, 0), v100, z5, tool0;
MoveL Offs(p0,88.596,280.02160000000003, 0), v100, z5, tool0;
MoveL Offs(p0,88.836,284.1917, 0), v100, z5, tool0;
MoveL Offs(p0,88.8,288.0, 0), v100, z5, tool0;
MoveL Offs(p0,88.5057,292.014, 0), v100, z5, tool0;
MoveL Offs(p0,88.3664,292.856, 0), v100, z5, tool0;
MoveL Offs(p0,88.1875,293.5, 0), v100, z5, tool0;
MoveL Offs(p0,87.9576,293.976, 0), v100, z5, tool0;
MoveL Offs(p0,87.6653,294.314, 0), v100, z5, tool0;
MoveL Offs(p0,87.29920000000001,294.54400000000004, 0), v100, z5, tool0;
MoveL Offs(p0,86.84790000000001,294.696, 0), v100, z5, tool0;
MoveL Offs(p0,86.3,294.8, 0), v100, z5, tool0;
MoveL Offs(p0,84.5832,294.5968, 0), v100, z5, tool0;
MoveL Offs(p0,84.3625,294.2625, 0), v100, z5, tool0;
MoveL Offs(p0,84.2048,293.7632, 0), v100, z5, tool0;
MoveL Offs(p0,84.0999,293.07309999999995, 0), v100, z5, tool0;
MoveL Offs(p0,84.0376,292.1664, 0), v100, z5, tool0;
MoveL Offs(p0,84.00770000000001,291.01730000000003, 0), v100, z5, tool0;
MoveL Offs(p0,84.0,289.6, 0), v100, z5, tool0;
MoveL Offs(p0,83.65979999999999,285.1621, 0), v100, z5, tool0;
MoveL Offs(p0,83.4016,284.3152, 0), v100, z5, tool0;
MoveL Offs(p0,83.075,283.7875, 0), v100, z5, tool0;
MoveL Offs(p0,82.6824,283.5808, 0), v100, z5, tool0;
MoveL Offs(p0,82.22619999999999,283.6969, 0), v100, z5, tool0;
MoveL Offs(p0,81.7088,284.1376, 0), v100, z5, tool0;
MoveL Offs(p0,81.1326,284.9047, 0), v100, z5, tool0;
MoveL Offs(p0,80.5,286.0, 0), v100, z5, tool0;
MoveL Offs(p0,80.0095,286.92760000000004, 0), v100, z5, tool0;
MoveL Offs(p0,79.55200000000002,287.6728000000001, 0), v100, z5, tool0;
MoveL Offs(p0,79.1185,288.2392, 0), v100, z5, tool0;
MoveL Offs(p0,78.70000000000002,288.6304, 0), v100, z5, tool0;
MoveL Offs(p0,78.2875,288.85, 0), v100, z5, tool0;
MoveL Offs(p0,77.872,288.90160000000003, 0), v100, z5, tool0;
MoveL Offs(p0,77.44449999999999,288.7888, 0), v100, z5, tool0;
MoveL Offs(p0,76.99600000000001,288.51520000000005, 0), v100, z5, tool0;
MoveL Offs(p0,76.51750000000001,288.0844, 0), v100, z5, tool0;
MoveL Offs(p0,76.0,287.5, 0), v100, z5, tool0;
MoveL Offs(p0,75.6614,287.1254, 0), v100, z5, tool0;
MoveL Offs(p0,75.35520000000001,286.8432000000001, 0), v100, z5, tool0;
MoveL Offs(p0,75.0658,286.6558, 0), v100, z5, tool0;
MoveL Offs(p0,74.77759999999999,286.5656, 0), v100, z5, tool0;
MoveL Offs(p0,74.475,286.575, 0), v100, z5, tool0;
MoveL Offs(p0,74.14240000000001,286.6864, 0), v100, z5, tool0;
MoveL Offs(p0,73.76419999999999,286.9022, 0), v100, z5, tool0;
MoveL Offs(p0,73.32480000000001,287.2248000000001, 0), v100, z5, tool0;
MoveL Offs(p0,72.2,288.2, 0), v100, z5, tool0;
MoveL Offs(p0,69.8,290.5, 0), v100, z5, tool0;
MoveL Offs(p0,68.3,288.3, 0), v100, z5, tool0;
MoveL Offs(p0,68.02770000000001,287.91970000000003, 0), v100, z5, tool0;
MoveL Offs(p0,67.75360000000002,287.5616000000001, 0), v100, z5, tool0;
MoveL Offs(p0,67.4819,287.2299, 0), v100, z5, tool0;
MoveL Offs(p0,67.2168,286.9288, 0), v100, z5, tool0;
MoveL Offs(p0,66.9625,286.6625, 0), v100, z5, tool0;
MoveL Offs(p0,66.72319999999999,286.4352, 0), v100, z5, tool0;
MoveL Offs(p0,66.50309999999999,286.2511, 0), v100, z5, tool0;
MoveL Offs(p0,66.30640000000001,286.11440000000005, 0), v100, z5, tool0;
MoveL Offs(p0,66.13730000000001,286.0293, 0), v100, z5, tool0;
MoveL Offs(p0,66.0,286.0, 0), v100, z5, tool0;
MoveL Offs(p0,65.66000000000003,286.2968, 0), v100, z5, tool0;
MoveL Offs(p0,65.424,286.65070000000003, 0), v100, z5, tool0;
MoveL Offs(p0,65.152,287.1264, 0), v100, z5, tool0;
MoveL Offs(p0,64.85,287.7125, 0), v100, z5, tool0;
MoveL Offs(p0,64.524,288.3976, 0), v100, z5, tool0;
MoveL Offs(p0,64.17999999999999,289.1703, 0), v100, z5, tool0;
MoveL Offs(p0,63.824,290.0192, 0), v100, z5, tool0;
MoveL Offs(p0,63.462,290.9329, 0), v100, z5, tool0;
MoveL Offs(p0,63.1,291.9, 0), v100, z5, tool0;
MoveL Offs(p0,62.31700000000001,293.9538000000001, 0), v100, z5, tool0;
MoveL Offs(p0,61.480000000000004,295.8984000000001, 0), v100, z5, tool0;
MoveL Offs(p0,60.60699999999999,297.70860000000005, 0), v100, z5, tool0;
MoveL Offs(p0,59.71600000000001,299.3592, 0), v100, z5, tool0;
MoveL Offs(p0,58.825,300.825, 0), v100, z5, tool0;
MoveL Offs(p0,57.952,302.0808, 0), v100, z5, tool0;
MoveL Offs(p0,57.114999999999995,303.1014, 0), v100, z5, tool0;
MoveL Offs(p0,56.33200000000001,303.8616, 0), v100, z5, tool0;
MoveL Offs(p0,55.621,304.3362, 0), v100, z5, tool0;
MoveL Offs(p0,55.0,304.5, 0), v100, z5, tool0;
MoveL Offs(p0,53.999199999999995,304.87260000000003, 0), v100, z5, tool0;
MoveL Offs(p0,53.5664,305.14320000000004, 0), v100, z5, tool0;
MoveL Offs(p0,53.1,305.475, 0), v100, z5, tool0;
MoveL Offs(p0,52.6096,305.86080000000004, 0), v100, z5, tool0;
MoveL Offs(p0,52.1048,306.2934, 0), v100, z5, tool0;
MoveL Offs(p0,51.5952,306.7656, 0), v100, z5, tool0;
MoveL Offs(p0,51.0904,307.27020000000005, 0), v100, z5, tool0;
MoveL Offs(p0,50.6,307.8, 0), v100, z5, tool0;
MoveL Offs(p0,49.6619,308.768, 0), v100, z5, tool0;
MoveL Offs(p0,48.723200000000006,309.56800000000004, 0), v100, z5, tool0;
MoveL Offs(p0,47.8073,310.19399999999996, 0), v100, z5, tool0;
MoveL Offs(p0,46.9376,310.64, 0), v100, z5, tool0;
MoveL Offs(p0,46.1375,310.9, 0), v100, z5, tool0;
MoveL Offs(p0,45.4304,310.96799999999996, 0), v100, z5, tool0;
MoveL Offs(p0,44.83970000000001,310.838, 0), v100, z5, tool0;
MoveL Offs(p0,44.3888,310.504, 0), v100, z5, tool0;
MoveL Offs(p0,44.1011,309.96000000000004, 0), v100, z5, tool0;
MoveL Offs(p0,44.0,309.2, 0), v100, z5, tool0;
MoveL Offs(p0,44.275,307.0375, 0), v100, z5, tool0;
MoveL Offs(p0,44.388799999999996,306.47839999999997, 0), v100, z5, tool0;
MoveL Offs(p0,44.5194,305.9037, 0), v100, z5, tool0;
MoveL Offs(p0,44.665600000000005,305.32480000000004, 0), v100, z5, tool0;
MoveL Offs(p0,44.82620000000001,304.7531, 0), v100, z5, tool0;
MoveL Offs(p0,45.0,304.2, 0), v100, z5, tool0;
MoveL Offs(p0,45.2128,303.40670000000006, 0), v100, z5, tool0;
MoveL Offs(p0,45.37040000000001,302.7616000000001, 0), v100, z5, tool0;
MoveL Offs(p0,45.4716,302.2569, 0), v100, z5, tool0;
MoveL Offs(p0,45.51520000000001,301.88480000000004, 0), v100, z5, tool0;
MoveL Offs(p0,45.5,301.6375, 0), v100, z5, tool0;
MoveL Offs(p0,45.4248,301.50719999999995, 0), v100, z5, tool0;
MoveL Offs(p0,45.2884,301.48609999999996, 0), v100, z5, tool0;
MoveL Offs(p0,44.5,302.0, 0), v100, z5, tool0;
MoveL Offs(p0,43.77460000000001,302.53240000000005, 0), v100, z5, tool0;
MoveL Offs(p0,43.16080000000001,302.8152000000001, 0), v100, z5, tool0;
MoveL Offs(p0,42.6622,302.85679999999996, 0), v100, z5, tool0;
MoveL Offs(p0,42.2824,302.66560000000004, 0), v100, z5, tool0;
MoveL Offs(p0,42.025,302.25, 0), v100, z5, tool0;
MoveL Offs(p0,41.8936,301.61839999999995, 0), v100, z5, tool0;
MoveL Offs(p0,41.8918,300.7792, 0), v100, z5, tool0;
MoveL Offs(p0,42.02320000000001,299.74080000000004, 0), v100, z5, tool0;
MoveL Offs(p0,42.291399999999996,298.51160000000004, 0), v100, z5, tool0;
MoveL Offs(p0,42.7,297.1, 0), v100, z5, tool0;
MoveL Offs(p0,42.954699999999995,296.2833, 0), v100, z5, tool0;
MoveL Offs(p0,43.17760000000001,295.46240000000006, 0), v100, z5, tool0;
MoveL Offs(p0,43.3669,294.6511, 0), v100, z5, tool0;
MoveL Offs(p0,43.5208,293.86320000000006, 0), v100, z5, tool0;
MoveL Offs(p0,43.6375,293.1125, 0), v100, z5, tool0;
MoveL Offs(p0,43.715199999999996,292.41279999999995, 0), v100, z5, tool0;
MoveL Offs(p0,43.7521,291.7779, 0), v100, z5, tool0;
MoveL Offs(p0,43.74640000000001,291.2216, 0), v100, z5, tool0;
MoveL Offs(p0,43.6963,290.7577, 0), v100, z5, tool0;
MoveL Offs(p0,43.6,290.4, 0), v100, z5, tool0;
MoveL Offs(p0,43.22800000000001,289.6128000000001, 0), v100, z5, tool0;
MoveL Offs(p0,43.064499999999995,289.39919999999995, 0), v100, z5, tool0;
MoveL Offs(p0,42.904,289.3104000000001, 0), v100, z5, tool0;
MoveL Offs(p0,42.7375,289.35, 0), v100, z5, tool0;
MoveL Offs(p0,42.556,289.5216, 0), v100, z5, tool0;
MoveL Offs(p0,42.3505,289.8288, 0), v100, z5, tool0;
MoveL Offs(p0,41.8315,290.86440000000005, 0), v100, z5, tool0;
MoveL Offs(p0,41.5,291.6, 0), v100, z5, tool0;
MoveL Offs(p0,40.952000000000005,292.82430000000005, 0), v100, z5, tool0;
MoveL Offs(p0,40.44000000000001,293.7984, 0), v100, z5, tool0;
MoveL Offs(p0,39.952,294.5241, 0), v100, z5, tool0;
MoveL Offs(p0,39.476,295.0032, 0), v100, z5, tool0;
MoveL Offs(p0,39.0,295.2375, 0), v100, z5, tool0;
MoveL Offs(p0,38.512,295.2288, 0), v100, z5, tool0;
MoveL Offs(p0,38.0,294.97889999999995, 0), v100, z5, tool0;
MoveL Offs(p0,37.452000000000005,294.4896, 0), v100, z5, tool0;
MoveL Offs(p0,36.856,293.7627, 0), v100, z5, tool0;
MoveL Offs(p0,36.2,292.8, 0), v100, z5, tool0;
MoveL Offs(p0,34.2,289.7, 0), v100, z5, tool0;
MoveL Offs(p0,32.6,292.8, 0), v100, z5, tool0;
MoveL Offs(p0,32.32490000000001,293.32700000000006, 0), v100, z5, tool0;
MoveL Offs(p0,32.04320000000001,293.824, 0), v100, z5, tool0;
MoveL Offs(p0,31.760299999999994,294.28499999999997, 0), v100, z5, tool0;
MoveL Offs(p0,31.481600000000004,294.70400000000006, 0), v100, z5, tool0;
MoveL Offs(p0,31.2125,295.075, 0), v100, z5, tool0;
MoveL Offs(p0,30.9584,295.392, 0), v100, z5, tool0;
MoveL Offs(p0,30.724700000000002,295.649, 0), v100, z5, tool0;
MoveL Offs(p0,30.5168,295.84000000000003, 0), v100, z5, tool0;
MoveL Offs(p0,30.3401,295.959, 0), v100, z5, tool0;
MoveL Offs(p0,30.2,296.0, 0), v100, z5, tool0;
MoveL Offs(p0,29.606900000000003,295.5787999999999, 0), v100, z5, tool0;
MoveL Offs(p0,29.3568,295.27360000000004, 0), v100, z5, tool0;
MoveL Offs(p0,29.0875,294.9, 0), v100, z5, tool0;
MoveL Offs(p0,28.803199999999997,294.46639999999996, 0), v100, z5, tool0;
MoveL Offs(p0,28.508099999999995,293.9812, 0), v100, z5, tool0;
MoveL Offs(p0,28.206400000000002,293.4528, 0), v100, z5, tool0;
MoveL Offs(p0,27.902300000000004,292.88960000000003, 0), v100, z5, tool0;
MoveL Offs(p0,27.6,292.3, 0), v100, z5, tool0;
MoveL Offs(p0,27.132400000000008,291.35040000000004, 0), v100, z5, tool0;
MoveL Offs(p0,26.73920000000001,290.5952000000001, 0), v100, z5, tool0;
MoveL Offs(p0,26.4048,290.02479999999997, 0), v100, z5, tool0;
MoveL Offs(p0,26.1136,289.6296000000001, 0), v100, z5, tool0;
MoveL Offs(p0,25.85,289.4, 0), v100, z5, tool0;
MoveL Offs(p0,25.5984,289.32640000000004, 0), v100, z5, tool0;
MoveL Offs(p0,25.343200000000003,289.39919999999995, 0), v100, z5, tool0;
MoveL Offs(p0,25.068800000000003,289.60880000000003, 0), v100, z5, tool0;
MoveL Offs(p0,24.7596,289.9456, 0), v100, z5, tool0;
MoveL Offs(p0,24.4,290.4, 0), v100, z5, tool0;
MoveL Offs(p0,24.187700000000003,290.71080000000006, 0), v100, z5, tool0;
MoveL Offs(p0,23.973600000000005,291.0384000000001, 0), v100, z5, tool0;
MoveL Offs(p0,23.761899999999997,291.37559999999996, 0), v100, z5, tool0;
MoveL Offs(p0,23.556800000000003,291.7152, 0), v100, z5, tool0;
MoveL Offs(p0,23.3625,292.05, 0), v100, z5, tool0;
MoveL Offs(p0,23.1832,292.3728, 0), v100, z5, tool0;
MoveL Offs(p0,23.0231,292.67639999999994, 0), v100, z5, tool0;
MoveL Offs(p0,22.886400000000002,292.9536, 0), v100, z5, tool0;
MoveL Offs(p0,22.777300000000004,293.1972, 0), v100, z5, tool0;
MoveL Offs(p0,22.7,293.4, 0), v100, z5, tool0;
MoveL Offs(p0,22.492800000000006,293.7728000000001, 0), v100, z5, tool0;
MoveL Offs(p0,22.3652,293.8797, 0), v100, z5, tool0;
MoveL Offs(p0,22.218400000000003,293.93440000000004, 0), v100, z5, tool0;
MoveL Offs(p0,22.05,293.9375, 0), v100, z5, tool0;
MoveL Offs(p0,21.857599999999998,293.88960000000003, 0), v100, z5, tool0;
MoveL Offs(p0,21.6388,293.7913, 0), v100, z5, tool0;
MoveL Offs(p0,21.391200000000005,293.6432000000001, 0), v100, z5, tool0;
MoveL Offs(p0,20.8,293.2, 0), v100, z5, tool0;
MoveL Offs(p0,20.436,292.90970000000004, 0), v100, z5, tool0;
MoveL Offs(p0,20.120000000000005,292.7016000000001, 0), v100, z5, tool0;
MoveL Offs(p0,19.845999999999997,292.57989999999995, 0), v100, z5, tool0;
MoveL Offs(p0,19.608,292.54879999999997, 0), v100, z5, tool0;
MoveL Offs(p0,19.4,292.6125, 0), v100, z5, tool0;
MoveL Offs(p0,19.216,292.7752, 0), v100, z5, tool0;
MoveL Offs(p0,18.896000000000004,293.4144, 0), v100, z5, tool0;
MoveL Offs(p0,18.748,293.8993, 0), v100, z5, tool0;
MoveL Offs(p0,18.6,294.5, 0), v100, z5, tool0;
MoveL Offs(p0,18.299200000000006,295.41280000000006, 0), v100, z5, tool0;
MoveL Offs(p0,18.1023,295.7896999999999, 0), v100, z5, tool0;
MoveL Offs(p0,17.873600000000003,296.11440000000005, 0), v100, z5, tool0;
MoveL Offs(p0,17.6125,296.3875, 0), v100, z5, tool0;
MoveL Offs(p0,17.3184,296.6096, 0), v100, z5, tool0;
MoveL Offs(p0,16.9907,296.7813, 0), v100, z5, tool0;
MoveL Offs(p0,16.628800000000002,296.9032, 0), v100, z5, tool0;
MoveL Offs(p0,16.2321,296.9759, 0), v100, z5, tool0;
MoveL Offs(p0,15.8,297.0, 0), v100, z5, tool0;
MoveL Offs(p0,14.480599999999999,296.7353999999999, 0), v100, z5, tool0;
MoveL Offs(p0,14.2352,296.4208, 0), v100, z5, tool0;
MoveL Offs(p0,14.075,295.925, 0), v100, z5, tool0;
MoveL Offs(p0,13.992799999999999,295.20719999999994, 0), v100, z5, tool0;
MoveL Offs(p0,13.981399999999999,294.22659999999996, 0), v100, z5, tool0;
MoveL Offs(p0,14.033600000000002,292.9424, 0), v100, z5, tool0;
MoveL Offs(p0,14.142200000000003,291.3138, 0), v100, z5, tool0;
MoveL Offs(p0,14.3,289.3, 0), v100, z5, tool0;
MoveL Offs(p0,14.804700000000002,284.8038000000001, 0), v100, z5, tool0;
MoveL Offs(p0,15.589600000000008,280.1624000000001, 0), v100, z5, tool0;
MoveL Offs(p0,16.640900000000002,275.41659999999996, 0), v100, z5, tool0;
MoveL Offs(p0,17.9448,270.60720000000003, 0), v100, z5, tool0;
MoveL Offs(p0,19.4875,265.775, 0), v100, z5, tool0;
MoveL Offs(p0,21.255200000000002,260.9608, 0), v100, z5, tool0;
MoveL Offs(p0,23.2341,256.2054, 0), v100, z5, tool0;
MoveL Offs(p0,25.410400000000003,251.5496, 0), v100, z5, tool0;
MoveL Offs(p0,27.770300000000002,247.0342, 0), v100, z5, tool0;
MoveL Offs(p0,30.3,242.7, 0), v100, z5, tool0;
MoveL Offs(p0,32.29610000000001,239.4632, 0), v100, z5, tool0;
MoveL Offs(p0,33.86080000000001,236.8936000000001, 0), v100, z5, tool0;
MoveL Offs(p0,35.0187,234.90240000000003, 0), v100, z5, tool0;
MoveL Offs(p0,35.7944,233.40080000000006, 0), v100, z5, tool0;
MoveL Offs(p0,36.2125,232.3, 0), v100, z5, tool0;
MoveL Offs(p0,36.2976,231.5112, 0), v100, z5, tool0;
MoveL Offs(p0,36.0743,230.9456, 0), v100, z5, tool0;
MoveL Offs(p0,35.5672,230.51440000000002, 0), v100, z5, tool0;
MoveL Offs(p0,34.8009,230.1288, 0), v100, z5, tool0;
MoveL Offs(p0,33.8,229.7, 0), v100, z5, tool0;
MoveL Offs(p0,31.5896,228.52090000000004, 0), v100, z5, tool0;
MoveL Offs(p0,29.472800000000007,226.92720000000008, 0), v100, z5, tool0;
MoveL Offs(p0,27.4712,224.95430000000002, 0), v100, z5, tool0;
MoveL Offs(p0,25.606400000000008,222.63760000000002, 0), v100, z5, tool0;
MoveL Offs(p0,23.9,220.0125, 0), v100, z5, tool0;
MoveL Offs(p0,22.3736,217.11440000000002, 0), v100, z5, tool0;
MoveL Offs(p0,21.048799999999996,213.97869999999998, 0), v100, z5, tool0;
MoveL Offs(p0,19.947200000000002,210.64080000000004, 0), v100, z5, tool0;
MoveL Offs(p0,19.0904,207.1361, 0), v100, z5, tool0;
MoveL Offs(p0,18.5,203.5, 0), v100, z5, tool0;
MoveL Offs(p0,18.110400000000006,201.09520000000003, 0), v100, z5, tool0;
MoveL Offs(p0,17.887100000000004,200.09529999999998, 0), v100, z5, tool0;
MoveL Offs(p0,17.6392,199.21359999999999, 0), v100, z5, tool0;
MoveL Offs(p0,17.3625,198.4375, 0), v100, z5, tool0;
MoveL Offs(p0,17.052799999999998,197.7544, 0), v100, z5, tool0;
MoveL Offs(p0,16.7059,197.1517, 0), v100, z5, tool0;
MoveL Offs(p0,16.317600000000002,196.6168, 0), v100, z5, tool0;
MoveL Offs(p0,15.883700000000001,196.1371, 0), v100, z5, tool0;
MoveL Offs(p0,15.4,195.7, 0), v100, z5, tool0;
MoveL Offs(p0,14.970000000000002,195.30720000000002, 0), v100, z5, tool0;
MoveL Offs(p0,14.468000000000004,194.74160000000006, 0), v100, z5, tool0;
MoveL Offs(p0,13.905999999999997,194.02239999999998, 0), v100, z5, tool0;
MoveL Offs(p0,13.296000000000001,193.1688, 0), v100, z5, tool0;
MoveL Offs(p0,12.65,192.2, 0), v100, z5, tool0;
MoveL Offs(p0,11.98,191.1352, 0), v100, z5, tool0;
MoveL Offs(p0,11.297999999999998,189.99359999999996, 0), v100, z5, tool0;
MoveL Offs(p0,10.616000000000001,188.7944, 0), v100, z5, tool0;
MoveL Offs(p0,9.946000000000002,187.5568, 0), v100, z5, tool0;
MoveL Offs(p0,9.3,186.3, 0), v100, z5, tool0;
MoveL Offs(p0,8.3186,184.26440000000002, 0), v100, z5, tool0;
MoveL Offs(p0,7.520800000000003,182.53120000000004, 0), v100, z5, tool0;
MoveL Offs(p0,6.8862,181.00079999999997, 0), v100, z5, tool0;
MoveL Offs(p0,6.394400000000001,179.57360000000003, 0), v100, z5, tool0;
MoveL Offs(p0,6.025,178.15, 0), v100, z5, tool0;
MoveL Offs(p0,5.7576,176.6304, 0), v100, z5, tool0;
MoveL Offs(p0,5.5718000000000005,174.9152, 0), v100, z5, tool0;
MoveL Offs(p0,5.4472000000000005,172.90480000000002, 0), v100, z5, tool0;
MoveL Offs(p0,5.3634,170.49960000000002, 0), v100, z5, tool0;
MoveL Offs(p0,5.3,167.6, 0), v100, z5, tool0;
MoveL Offs(p0,5.077699999999999,160.8842, 0), v100, z5, tool0;
MoveL Offs(p0,4.930400000000001,159.1824, 0), v100, z5, tool0;
MoveL Offs(p0,4.7375,157.675, 0), v100, z5, tool0;
MoveL Offs(p0,4.4936,156.3176, 0), v100, z5, tool0;
MoveL Offs(p0,4.1933,155.0658, 0), v100, z5, tool0;
MoveL Offs(p0,3.8312000000000004,153.8752, 0), v100, z5, tool0;
MoveL Offs(p0,3.4019,152.7014, 0), v100, z5, tool0;
MoveL Offs(p0,2.9,151.5, 0), v100, z5, tool0;
MoveL Offs(p0,1.9675,148.97350000000003, 0), v100, z5, tool0;
MoveL Offs(p0,1.2120000000000002,145.96400000000003, 0), v100, z5, tool0;
MoveL Offs(p0,0.6364999999999996,142.57649999999998, 0), v100, z5, tool0;
MoveL Offs(p0,0.2439999999999999,138.916, 0), v100, z5, tool0;
MoveL Offs(p0,0.0375,135.0875, 0), v100, z5, tool0;
MoveL Offs(p0,0.020000000000000108,131.196, 0), v100, z5, tool0;
MoveL Offs(p0,0.19450000000000012,127.34649999999999, 0), v100, z5, tool0;
MoveL Offs(p0,0.5640000000000002,123.644, 0), v100, z5, tool0;
MoveL Offs(p0,1.1315000000000004,120.1935, 0), v100, z5, tool0;
MoveL Offs(p0,1.9,117.1, 0), v100, z5, tool0;
MoveL Offs(p0,2.2504000000000004,115.922, 0), v100, z5, tool0;
MoveL Offs(p0,2.5792000000000006,114.68400000000004, 0), v100, z5, tool0;
MoveL Offs(p0,2.8828000000000005,113.41, 0), v100, z5, tool0;
MoveL Offs(p0,3.157600000000001,112.124, 0), v100, z5, tool0;
MoveL Offs(p0,3.4,110.85, 0), v100, z5, tool0;
MoveL Offs(p0,3.6064000000000007,109.612, 0), v100, z5, tool0;
MoveL Offs(p0,3.7732,108.434, 0), v100, z5, tool0;
MoveL Offs(p0,3.8968000000000003,107.34, 0), v100, z5, tool0;
MoveL Offs(p0,3.9736000000000002,106.354, 0), v100, z5, tool0;
MoveL Offs(p0,4.0,105.5, 0), v100, z5, tool0;
MoveL Offs(p0,4.442400000000001,101.61600000000001, 0), v100, z5, tool0;
MoveL Offs(p0,4.953100000000001,99.1955, 0), v100, z5, tool0;
MoveL Offs(p0,5.619200000000001,96.58000000000001, 0), v100, z5, tool0;
MoveL Offs(p0,6.4125,93.8625, 0), v100, z5, tool0;
MoveL Offs(p0,7.304800000000002,91.136, 0), v100, z5, tool0;
MoveL Offs(p0,8.267900000000001,88.4935, 0), v100, z5, tool0;
MoveL Offs(p0,9.273600000000002,86.02799999999999, 0), v100, z5, tool0;
MoveL Offs(p0,10.293700000000001,83.83250000000001, 0), v100, z5, tool0;
MoveL Offs(p0,11.3,82.0, 0), v100, z5, tool0;
MoveL Offs(p0,11.6758,81.376, 0), v100, z5, tool0;
MoveL Offs(p0,12.134400000000005,80.65600000000003, 0), v100, z5, tool0;
MoveL Offs(p0,12.6626,79.85799999999999, 0), v100, z5, tool0;
MoveL Offs(p0,13.247200000000001,79.00000000000001, 0), v100, z5, tool0;
MoveL Offs(p0,13.875,78.1, 0), v100, z5, tool0;
MoveL Offs(p0,14.5328,77.176, 0), v100, z5, tool0;
MoveL Offs(p0,15.207399999999998,76.24600000000001, 0), v100, z5, tool0;
MoveL Offs(p0,15.885600000000002,75.328, 0), v100, z5, tool0;
MoveL Offs(p0,16.5542,74.44000000000001, 0), v100, z5, tool0;
MoveL Offs(p0,17.2,73.6, 0), v100, z5, tool0;
MoveL Offs(p0,17.816700000000004,72.78620000000002, 0), v100, z5, tool0;
MoveL Offs(p0,18.401600000000006,71.97360000000002, 0), v100, z5, tool0;
MoveL Offs(p0,18.9469,71.1754, 0), v100, z5, tool0;
MoveL Offs(p0,19.444799999999997,70.4048, 0), v100, z5, tool0;
MoveL Offs(p0,19.8875,69.675, 0), v100, z5, tool0;
MoveL Offs(p0,20.267199999999995,68.9992, 0), v100, z5, tool0;
MoveL Offs(p0,20.576100000000004,68.39059999999999, 0), v100, z5, tool0;
MoveL Offs(p0,20.806400000000004,67.86240000000001, 0), v100, z5, tool0;
MoveL Offs(p0,20.950300000000002,67.4278, 0), v100, z5, tool0;
MoveL Offs(p0,21.0,67.1, 0), v100, z5, tool0;
MoveL Offs(p0,21.326699999999995,65.6582, 0), v100, z5, tool0;
MoveL Offs(p0,21.566400000000005,64.93840000000002, 0), v100, z5, tool0;
MoveL Offs(p0,21.8625,64.125, 0), v100, z5, tool0;
MoveL Offs(p0,22.209600000000002,63.2336, 0), v100, z5, tool0;
MoveL Offs(p0,22.6023,62.2798, 0), v100, z5, tool0;
MoveL Offs(p0,23.035200000000003,61.27920000000002, 0), v100, z5, tool0;
MoveL Offs(p0,23.502900000000004,60.247400000000006, 0), v100, z5, tool0;
MoveL Offs(p0,24.0,59.2, 0), v100, z5, tool0;
MoveL Offs(p0,25.231900000000003,56.876400000000004, 0), v100, z5, tool0;
MoveL Offs(p0,26.739200000000004,54.495200000000025, 0), v100, z5, tool0;
MoveL Offs(p0,28.479299999999995,52.10079999999999, 0), v100, z5, tool0;
MoveL Offs(p0,30.4096,49.7376, 0), v100, z5, tool0;
MoveL Offs(p0,32.4875,47.45, 0), v100, z5, tool0;
MoveL Offs(p0,34.6704,45.282399999999996, 0), v100, z5, tool0;
MoveL Offs(p0,36.9157,43.279199999999996, 0), v100, z5, tool0;
MoveL Offs(p0,39.180800000000005,41.48480000000001, 0), v100, z5, tool0;
MoveL Offs(p0,41.423100000000005,39.9436, 0), v100, z5, tool0;
MoveL Offs(p0,43.6,38.7, 0), v100, z5, tool0;
MoveL Offs(p0,44.435100000000006,38.25750000000001, 0), v100, z5, tool0;
MoveL Offs(p0,45.252800000000015,37.77600000000001, 0), v100, z5, tool0;
MoveL Offs(p0,46.041700000000006,37.26449999999999, 0), v100, z5, tool0;
MoveL Offs(p0,46.790400000000005,36.732000000000006, 0), v100, z5, tool0;
MoveL Offs(p0,47.4875,36.1875, 0), v100, z5, tool0;
MoveL Offs(p0,48.121599999999994,35.64, 0), v100, z5, tool0;
MoveL Offs(p0,48.6813,35.0985, 0), v100, z5, tool0;
MoveL Offs(p0,49.1552,34.572, 0), v100, z5, tool0;
MoveL Offs(p0,49.5319,34.0695, 0), v100, z5, tool0;
MoveL Offs(p0,49.8,33.6, 0), v100, z5, tool0;
MoveL Offs(p0,51.49670000000001,30.6313, 0), v100, z5, tool0;
MoveL Offs(p0,53.88160000000001,27.64640000000001, 0), v100, z5, tool0;
MoveL Offs(p0,56.856899999999996,24.707099999999997, 0), v100, z5, tool0;
MoveL Offs(p0,60.3248,21.8752, 0), v100, z5, tool0;
MoveL Offs(p0,64.1875,19.2125, 0), v100, z5, tool0;
MoveL Offs(p0,68.3472,16.7808, 0), v100, z5, tool0;
MoveL Offs(p0,72.7061,14.641899999999998, 0), v100, z5, tool0;
MoveL Offs(p0,77.16640000000001,12.8576, 0), v100, z5, tool0;
MoveL Offs(p0,81.6303,11.489700000000001, 0), v100, z5, tool0;
MoveL Offs(p0,86.0,10.6, 0), v100, z5, tool0;
MoveL Offs(p0,87.79120000000002,10.192000000000004, 0), v100, z5, tool0;
MoveL Offs(p0,88.8683,9.875499999999999, 0), v100, z5, tool0;
MoveL Offs(p0,90.0336,9.496, 0), v100, z5, tool0;
MoveL Offs(p0,91.2625,9.0625, 0), v100, z5, tool0;
MoveL Offs(p0,92.53040000000001,8.584, 0), v100, z5, tool0;
MoveL Offs(p0,93.81269999999999,8.0695, 0), v100, z5, tool0;
MoveL Offs(p0,95.0848,7.5280000000000005, 0), v100, z5, tool0;
MoveL Offs(p0,96.3221,6.968500000000001, 0), v100, z5, tool0;
MoveL Offs(p0,97.5,6.4, 0), v100, z5, tool0;
MoveL Offs(p0,100.6932,4.9008, 0), v100, z5, tool0;
MoveL Offs(p0,103.71360000000001,3.6344000000000016, 0), v100, z5, tool0;
MoveL Offs(p0,106.62239999999997,2.5875999999999992, 0), v100, z5, tool0;
MoveL Offs(p0,109.4808,1.7471999999999999, 0), v100, z5, tool0;
MoveL Offs(p0,112.35,1.1, 0), v100, z5, tool0;
MoveL Offs(p0,115.2912,0.6327999999999997, 0), v100, z5, tool0;
MoveL Offs(p0,118.3656,0.33239999999999986, 0), v100, z5, tool0;
MoveL Offs(p0,121.6344,0.18559999999999996, 0), v100, z5, tool0;
MoveL Offs(p0,125.1588,0.17920000000000003, 0), v100, z5, tool0;
MoveL Offs(p0,129.0,0.3, 0), v100, z5, tool0;
MoveL Offs(p0,133.06560000000002,0.5480000000000002, 0), v100, z5, tool0;
MoveL Offs(p0,135.01289999999997,0.7185, 0), v100, z5, tool0;
MoveL Offs(p0,136.87680000000003,0.916, 0), v100, z5, tool0;
MoveL Offs(p0,138.6375,1.1375, 0), v100, z5, tool0;
MoveL Offs(p0,140.27519999999998,1.3800000000000001, 0), v100, z5, tool0;
MoveL Offs(p0,141.7701,1.6405, 0), v100, z5, tool0;
MoveL Offs(p0,143.10240000000002,1.9160000000000004, 0), v100, z5, tool0;
MoveL Offs(p0,144.2523,2.2035, 0), v100, z5, tool0;
MoveL Offs(p0,145.2,2.5, 0), v100, z5, tool0;
MoveL Offs(p0,146.37130000000002,2.9056, 0), v100, z5, tool0;
MoveL Offs(p0,147.45440000000002,3.2248000000000006, 0), v100, z5, tool0;
MoveL Offs(p0,148.49309999999997,3.4612000000000003, 0), v100, z5, tool0;
MoveL Offs(p0,149.5312,3.6184000000000003, 0), v100, z5, tool0;
MoveL Offs(p0,150.6125,3.7, 0), v100, z5, tool0;
MoveL Offs(p0,151.7808,3.7096000000000005, 0), v100, z5, tool0;
MoveL Offs(p0,153.0799,3.6507999999999994, 0), v100, z5, tool0;
MoveL Offs(p0,154.55360000000002,3.5272000000000006, 0), v100, z5, tool0;
MoveL Offs(p0,156.2457,3.3424, 0), v100, z5, tool0;
MoveL Offs(p0,158.2,3.1, 0), v100, z5, tool0;
MoveL Offs(p0,166.15030000000002,2.5669000000000004, 0), v100, z5, tool0;
MoveL Offs(p0,182.1661,4.4023, 0), v100, z5, tool0;
MoveL Offs(p0,189.9472,6.637600000000001, 0), v100, z5, tool0;
MoveL Offs(p0,197.3875,9.6625, 0), v100, z5, tool0;
MoveL Offs(p0,204.34480000000002,13.410400000000005, 0), v100, z5, tool0;
MoveL Offs(p0,210.67690000000002,17.814700000000006, 0), v100, z5, tool0;
MoveL Offs(p0,216.2416,22.808800000000005, 0), v100, z5, tool0;
MoveL Offs(p0,220.8967,28.326100000000004, 0), v100, z5, tool0;
MoveL Offs(p0,224.5,34.3, 0), v100, z5, tool0;
MoveL Offs(p0,225.1353,35.553200000000004, 0), v100, z5, tool0;
MoveL Offs(p0,225.74240000000003,36.63360000000001, 0), v100, z5, tool0;
MoveL Offs(p0,226.35309999999998,37.572399999999995, 0), v100, z5, tool0;
MoveL Offs(p0,226.99920000000003,38.400800000000004, 0), v100, z5, tool0;
MoveL Offs(p0,227.7125,39.15, 0), v100, z5, tool0;
MoveL Offs(p0,228.5248,39.8512, 0), v100, z5, tool0;
MoveL Offs(p0,229.46790000000001,40.5356, 0), v100, z5, tool0;
MoveL Offs(p0,230.5736,41.23440000000001, 0), v100, z5, tool0;
MoveL Offs(p0,231.8737,41.9788, 0), v100, z5, tool0;
MoveL Offs(p0,233.4,42.8, 0), v100, z5, tool0;
MoveL Offs(p0,237.61330000000007,45.36720000000001, 0), v100, z5, tool0;
MoveL Offs(p0,241.5824,48.51760000000001, 0), v100, z5, tool0;
MoveL Offs(p0,245.26109999999994,52.174400000000006, 0), v100, z5, tool0;
MoveL Offs(p0,248.60320000000002,56.2608, 0), v100, z5, tool0;
MoveL Offs(p0,251.5625,60.7, 0), v100, z5, tool0;
MoveL Offs(p0,254.09279999999998,65.4152, 0), v100, z5, tool0;
MoveL Offs(p0,256.14790000000005,70.3296, 0), v100, z5, tool0;
MoveL Offs(p0,257.6816,75.36640000000001, 0), v100, z5, tool0;
MoveL Offs(p0,258.6477,80.4488, 0), v100, z5, tool0;
MoveL Offs(p0,259.0,85.5, 0), v100, z5, tool0;
MoveL Offs(p0,259.26460000000003,88.0677, 0), v100, z5, tool0;
MoveL Offs(p0,259.4832,88.89840000000001, 0), v100, z5, tool0;
MoveL Offs(p0,259.775,89.7375, 0), v100, z5, tool0;
MoveL Offs(p0,260.14480000000003,90.5976, 0), v100, z5, tool0;
MoveL Offs(p0,260.5974,91.4913, 0), v100, z5, tool0;
MoveL Offs(p0,261.1376,92.43120000000002, 0), v100, z5, tool0;
MoveL Offs(p0,261.77020000000005,93.4299, 0), v100, z5, tool0;
MoveL Offs(p0,262.5,94.5, 0), v100, z5, tool0;
MoveL Offs(p0,264.33020000000005,97.42110000000001, 0), v100, z5, tool0;
MoveL Offs(p0,265.9696,100.73280000000003, 0), v100, z5, tool0;
MoveL Offs(p0,267.4014,104.3577, 0), v100, z5, tool0;
MoveL Offs(p0,268.60880000000003,108.21840000000002, 0), v100, z5, tool0;
MoveL Offs(p0,269.575,112.2375, 0), v100, z5, tool0;
MoveL Offs(p0,270.2832,116.3376, 0), v100, z5, tool0;
MoveL Offs(p0,270.7166,120.4413, 0), v100, z5, tool0;
MoveL Offs(p0,270.8584,124.4712, 0), v100, z5, tool0;
MoveL Offs(p0,270.6918,128.3499, 0), v100, z5, tool0;
MoveL Offs(p0,270.2,132.0, 0), v100, z5, tool0;
MoveL Offs(p0,269.87760000000014,133.74560000000002, 0), v100, z5, tool0;
MoveL Offs(p0,269.74639999999994,134.55689999999998, 0), v100, z5, tool0;
MoveL Offs(p0,269.6368,135.3088, 0), v100, z5, tool0;
MoveL Offs(p0,269.55,135.9875, 0), v100, z5, tool0;
MoveL Offs(p0,269.4872,136.5792, 0), v100, z5, tool0;
MoveL Offs(p0,269.44960000000003,137.0701, 0), v100, z5, tool0;
MoveL Offs(p0,269.4384,137.4464, 0), v100, z5, tool0;
MoveL Offs(p0,269.4548,137.6943, 0), v100, z5, tool0;
MoveL Offs(p0,269.5,137.8, 0), v100, z5, tool0;
MoveL Offs(p0,269.97120000000007,137.56560000000005, 0), v100, z5, tool0;
MoveL Offs(p0,270.4468,137.20239999999998, 0), v100, z5, tool0;
MoveL Offs(p0,271.0616,136.69279999999998, 0), v100, z5, tool0;
MoveL Offs(p0,271.8,136.05, 0), v100, z5, tool0;
MoveL Offs(p0,272.64639999999997,135.28719999999998, 0), v100, z5, tool0;
MoveL Offs(p0,273.5852,134.4176, 0), v100, z5, tool0;
MoveL Offs(p0,274.60080000000005,133.45440000000002, 0), v100, z5, tool0;
MoveL Offs(p0,275.6776,132.41080000000002, 0), v100, z5, tool0;
MoveL Offs(p0,276.8,131.3, 0), v100, z5, tool0;
MoveL Offs(p0,279.4227000000001,128.61260000000004, 0), v100, z5, tool0;
MoveL Offs(p0,281.9416000000001,125.78480000000005, 0), v100, z5, tool0;
MoveL Offs(p0,284.3429,122.8382, 0), v100, z5, tool0;
MoveL Offs(p0,286.6128,119.79440000000002, 0), v100, z5, tool0;
MoveL Offs(p0,288.7375,116.675, 0), v100, z5, tool0;
MoveL Offs(p0,290.70320000000004,113.50160000000001, 0), v100, z5, tool0;
MoveL Offs(p0,292.4961,110.29580000000001, 0), v100, z5, tool0;
MoveL Offs(p0,294.10240000000005,107.07920000000001, 0), v100, z5, tool0;
MoveL Offs(p0,295.5083,103.87339999999999, 0), v100, z5, tool0;
MoveL Offs(p0,296.7,100.7, 0), v100, z5, tool0;
MoveL Offs(p0,297.38590000000005,98.671, 0), v100, z5, tool0;
MoveL Offs(p0,297.9512000000001,96.85200000000003, 0), v100, z5, tool0;
MoveL Offs(p0,298.40729999999996,95.16499999999999, 0), v100, z5, tool0;
MoveL Offs(p0,298.7656,93.53200000000001, 0), v100, z5, tool0;
MoveL Offs(p0,299.0375,91.875, 0), v100, z5, tool0;
MoveL Offs(p0,299.2344,90.11600000000001, 0), v100, z5, tool0;
MoveL Offs(p0,299.3677,88.17699999999999, 0), v100, z5, tool0;
MoveL Offs(p0,299.4488,85.98, 0), v100, z5, tool0;
MoveL Offs(p0,299.48910000000006,83.447, 0), v100, z5, tool0;
MoveL Offs(p0,299.5,80.5, 0), v100, z5, tool0;
MoveL Offs(p0,299.23760000000004,71.2696, 0), v100, z5, tool0;
MoveL Offs(p0,299.0625,69.625, 0), v100, z5, tool0;
MoveL Offs(p0,298.8304,68.13039999999998, 0), v100, z5, tool0;
MoveL Offs(p0,298.5347,66.72819999999999, 0), v100, z5, tool0;
MoveL Offs(p0,298.16880000000003,65.3608, 0), v100, z5, tool0;
MoveL Offs(p0,297.7261,63.970600000000005, 0), v100, z5, tool0;
MoveL Offs(p0,297.2,62.5, 0), v100, z5, tool0;
MoveL Offs(p0,296.2439,60.14610000000001, 0), v100, z5, tool0;
MoveL Offs(p0,295.1792000000001,57.88880000000002, 0), v100, z5, tool0;
MoveL Offs(p0,294.0113,55.7347, 0), v100, z5, tool0;
MoveL Offs(p0,292.7456000000001,53.6904, 0), v100, z5, tool0;
MoveL Offs(p0,291.3875,51.7625, 0), v100, z5, tool0;
MoveL Offs(p0,289.9424,49.9576, 0), v100, z5, tool0;
MoveL Offs(p0,288.4157,48.2823, 0), v100, z5, tool0;
MoveL Offs(p0,286.81280000000004,46.7432, 0), v100, z5, tool0;
MoveL Offs(p0,285.1391,45.346900000000005, 0), v100, z5, tool0;
MoveL Offs(p0,283.4,44.1, 0), v100, z5, tool0;
MoveL Offs(p0,279.7945000000001,41.9731, 0), v100, z5, tool0;
MoveL Offs(p0,276.36,40.45280000000001, 0), v100, z5, tool0;
MoveL Offs(p0,273.0995,39.539699999999996, 0), v100, z5, tool0;
MoveL Offs(p0,270.01599999999996,39.2344, 0), v100, z5, tool0;
MoveL Offs(p0,267.1125,39.5375, 0), v100, z5, tool0;
MoveL Offs(p0,264.392,40.449600000000004, 0), v100, z5, tool0;
MoveL Offs(p0,261.85749999999996,41.9713, 0), v100, z5, tool0;
MoveL Offs(p0,257.3585,46.8459, 0), v100, z5, tool0;
MoveL Offs(p0,255.4,50.2, 0), v100, z5, tool0;
MoveL Offs(p0,254.87740000000008,51.18470000000001, 0), v100, z5, tool0;
MoveL Offs(p0,254.38720000000006,52.04160000000002, 0), v100, z5, tool0;
MoveL Offs(p0,253.92579999999998,52.7749, 0), v100, z5, tool0;
MoveL Offs(p0,253.48959999999997,53.3888, 0), v100, z5, tool0;
MoveL Offs(p0,253.075,53.8875, 0), v100, z5, tool0;
MoveL Offs(p0,252.67839999999995,54.2752, 0), v100, z5, tool0;
MoveL Offs(p0,252.2962,54.5561, 0), v100, z5, tool0;
MoveL Offs(p0,251.9248,54.73440000000001, 0), v100, z5, tool0;
MoveL Offs(p0,251.56060000000002,54.8143, 0), v100, z5, tool0;
MoveL Offs(p0,251.2,54.8, 0), v100, z5, tool0;
MoveL Offs(p0,250.49110000000002,54.4024, 0), v100, z5, tool0;
MoveL Offs(p0,249.98080000000004,53.61120000000002, 0), v100, z5, tool0;
MoveL Offs(p0,249.66369999999998,52.48879999999999, 0), v100, z5, tool0;
MoveL Offs(p0,249.5344,51.0976, 0), v100, z5, tool0;
MoveL Offs(p0,249.5875,49.5, 0), v100, z5, tool0;
MoveL Offs(p0,249.8176,47.758399999999995, 0), v100, z5, tool0;
MoveL Offs(p0,250.21930000000003,45.935199999999995, 0), v100, z5, tool0;
MoveL Offs(p0,250.78720000000004,44.0928, 0), v100, z5, tool0;
MoveL Offs(p0,251.51590000000002,42.293600000000005, 0), v100, z5, tool0;
MoveL Offs(p0,252.4,40.6, 0), v100, z5, tool0;
MoveL Offs(p0,253.97310000000007,38.227700000000006, 0), v100, z5, tool0;
MoveL Offs(p0,255.74480000000008,36.15360000000001, 0), v100, z5, tool0;
MoveL Offs(p0,257.70369999999997,34.3819, 0), v100, z5, tool0;
MoveL Offs(p0,259.8384,32.9168, 0), v100, z5, tool0;
MoveL Offs(p0,262.1375,31.7625, 0), v100, z5, tool0;
MoveL Offs(p0,264.5896,30.923199999999998, 0), v100, z5, tool0;
MoveL Offs(p0,267.18330000000003,30.403100000000002, 0), v100, z5, tool0;
MoveL Offs(p0,269.9072,30.206400000000002, 0), v100, z5, tool0;
MoveL Offs(p0,272.7499,30.337300000000006, 0), v100, z5, tool0;
MoveL Offs(p0,275.7,30.8, 0), v100, z5, tool0;
MoveL Offs(p0,280.80010000000004,32.17730000000001, 0), v100, z5, tool0;
MoveL Offs(p0,285.5888000000001,34.0784, 0), v100, z5, tool0;
MoveL Offs(p0,290.04869999999994,36.487100000000005, 0), v100, z5, tool0;
MoveL Offs(p0,294.16240000000005,39.3872, 0), v100, z5, tool0;
MoveL Offs(p0,297.9125,42.7625, 0), v100, z5, tool0;
MoveL Offs(p0,301.28159999999997,46.5968, 0), v100, z5, tool0;
MoveL Offs(p0,304.2523,50.873900000000006, 0), v100, z5, tool0;
MoveL Offs(p0,306.8072,55.577600000000004, 0), v100, z5, tool0;
MoveL Offs(p0,308.9289,60.691700000000004, 0), v100, z5, tool0;
MoveL Offs(p0,310.6,66.2, 0), v100, z5, tool0;
MoveL Offs(p0,311.27270000000004,69.41870000000002, 0), v100, z5, tool0;
MoveL Offs(p0,311.73360000000014,72.96560000000002, 0), v100, z5, tool0;
MoveL Offs(p0,311.9869,76.7669, 0), v100, z5, tool0;
MoveL Offs(p0,312.03679999999997,80.7488, 0), v100, z5, tool0;
MoveL Offs(p0,311.8875,84.8375, 0), v100, z5, tool0;
MoveL Offs(p0,311.5432,88.9592, 0), v100, z5, tool0;
MoveL Offs(p0,311.0081,93.04010000000001, 0), v100, z5, tool0;
MoveL Offs(p0,310.28640000000007,97.00640000000001, 0), v100, z5, tool0;
MoveL Offs(p0,309.3823,100.7843, 0), v100, z5, tool0;
MoveL Offs(p0,308.3,104.3, 0), v100, z5, tool0;
MoveL Offs(p0,306.3407,109.39460000000001, 0), v100, z5, tool0;
MoveL Offs(p0,304.06160000000006,114.36080000000001, 0), v100, z5, tool0;
MoveL Offs(p0,301.46090000000004,119.20219999999999, 0), v100, z5, tool0;
MoveL Offs(p0,298.5368,123.92240000000001, 0), v100, z5, tool0;
MoveL Offs(p0,295.2875,128.525, 0), v100, z5, tool0;
MoveL Offs(p0,291.7112,133.0136, 0), v100, z5, tool0;
MoveL Offs(p0,287.80609999999996,137.39180000000002, 0), v100, z5, tool0;
MoveL Offs(p0,283.5704,141.66320000000002, 0), v100, z5, tool0;
MoveL Offs(p0,279.0023,145.8314, 0), v100, z5, tool0;
MoveL Offs(p0,274.1,149.9, 0), v100, z5, tool0;
MoveL Offs(p0,265.3,156.8, 0), v100, z5, tool0;
MoveL Offs(p0,266.2,162.7, 0), v100, z5, tool0;
MoveL Offs(p0,266.4763,164.7399, 0), v100, z5, tool0;
MoveL Offs(p0,266.6464000000001,166.88720000000006, 0), v100, z5, tool0;
MoveL Offs(p0,266.7121,169.12330000000003, 0), v100, z5, tool0;
MoveL Offs(p0,266.6752,171.4296, 0), v100, z5, tool0;
MoveL Offs(p0,266.5375,173.7875, 0), v100, z5, tool0;
MoveL Offs(p0,265.9669,178.5837, 0), v100, z5, tool0;
MoveL Offs(p0,265.5376,180.9848, 0), v100, z5, tool0;
MoveL Offs(p0,265.01470000000006,183.3631, 0), v100, z5, tool0;
MoveL Offs(p0,264.4,185.7, 0), v100, z5, tool0;
MoveL Offs(p0,263.9771,187.21660000000003, 0), v100, z5, tool0;
MoveL Offs(p0,263.66880000000003,188.53280000000004, 0), v100, z5, tool0;
MoveL Offs(p0,263.4757,189.6582, 0), v100, z5, tool0;
MoveL Offs(p0,263.39840000000004,190.60240000000005, 0), v100, z5, tool0;
MoveL Offs(p0,263.4375,191.375, 0), v100, z5, tool0;
MoveL Offs(p0,263.5936,191.98559999999998, 0), v100, z5, tool0;
MoveL Offs(p0,263.8673,192.4438, 0), v100, z5, tool0;
MoveL Offs(p0,264.7699,192.94140000000002, 0), v100, z5, tool0;
MoveL Offs(p0,265.4,193.0, 0), v100, z5, tool0;
MoveL Offs(p0,266.11620000000005,192.5387, 0), v100, z5, tool0;
MoveL Offs(p0,267.22960000000006,191.18160000000006, 0), v100, z5, tool0;
MoveL Offs(p0,268.7174,188.96890000000002, 0), v100, z5, tool0;
MoveL Offs(p0,270.5568,185.94080000000002, 0), v100, z5, tool0;
MoveL Offs(p0,272.725,182.1375, 0), v100, z5, tool0;
MoveL Offs(p0,275.19919999999996,177.59919999999997, 0), v100, z5, tool0;
MoveL Offs(p0,277.9566,172.36610000000002, 0), v100, z5, tool0;
MoveL Offs(p0,280.97440000000006,166.47840000000002, 0), v100, z5, tool0;
MoveL Offs(p0,284.22979999999995,159.97629999999998, 0), v100, z5, tool0;
MoveL Offs(p0,287.7,152.9, 0), v100, z5, tool0;
MoveL Offs(p0,290.6492,146.92290000000003, 0), v100, z5, tool0;
MoveL Offs(p0,293.18560000000014,141.94720000000004, 0), v100, z5, tool0;
MoveL Offs(p0,295.3824,137.87629999999996, 0), v100, z5, tool0;
MoveL Offs(p0,297.31280000000004,134.61360000000002, 0), v100, z5, tool0;
MoveL Offs(p0,299.05,132.0625, 0), v100, z5, tool0;
MoveL Offs(p0,300.6672,130.1264, 0), v100, z5, tool0;
MoveL Offs(p0,302.23760000000004,128.7087, 0), v100, z5, tool0;
MoveL Offs(p0,303.8344,127.71280000000002, 0), v100, z5, tool0;
MoveL Offs(p0,305.5308,127.0421, 0), v100, z5, tool0;
MoveL Offs(p0,307.4,126.6, 0), v100, z5, tool0;
MoveL Offs(p0,313.4489,127.0752, 0), v100, z5, tool0;
MoveL Offs(p0,316.2208,127.8144, 0), v100, z5, tool0;
MoveL Offs(p0,319.3875,128.85, 0), v100, z5, tool0;
MoveL Offs(p0,322.95919999999995,130.1856, 0), v100, z5, tool0;
MoveL Offs(p0,326.9461,131.8248, 0), v100, z5, tool0;
MoveL Offs(p0,331.3584,133.7712, 0), v100, z5, tool0;
MoveL Offs(p0,336.2063,136.0284, 0), v100, z5, tool0;
MoveL Offs(p0,341.5,138.6, 0), v100, z5, tool0;
MoveL Offs(p0,347.04750000000007,141.39600000000002, 0), v100, z5, tool0;
MoveL Offs(p0,351.8000000000001,143.88000000000005, 0), v100, z5, tool0;
MoveL Offs(p0,355.8325,146.106, 0), v100, z5, tool0;
MoveL Offs(p0,359.21999999999997,148.128, 0), v100, z5, tool0;
MoveL Offs(p0,362.0375,150.0, 0), v100, z5, tool0;
MoveL Offs(p0,364.36,151.77599999999998, 0), v100, z5, tool0;
MoveL Offs(p0,366.2625,153.51, 0), v100, z5, tool0;
MoveL Offs(p0,367.82000000000005,155.256, 0), v100, z5, tool0;
MoveL Offs(p0,369.10749999999996,157.068, 0), v100, z5, tool0;
MoveL Offs(p0,370.2,159.0, 0), v100, z5, tool0;
MoveL Offs(p0,371.5522,161.82040000000003, 0), v100, z5, tool0;
MoveL Offs(p0,372.4376000000001,164.48720000000006, 0), v100, z5, tool0;
MoveL Offs(p0,372.7794,167.21880000000002, 0), v100, z5, tool0;
MoveL Offs(p0,372.5008,170.23360000000005, 0), v100, z5, tool0;
MoveL Offs(p0,371.525,173.75, 0), v100, z5, tool0;
MoveL Offs(p0,369.77520000000004,177.98639999999997, 0), v100, z5, tool0;
MoveL Offs(p0,367.1746,183.1612, 0), v100, z5, tool0;
MoveL Offs(p0,363.6464,189.49280000000002, 0), v100, z5, tool0;
MoveL Offs(p0,359.11379999999997,197.1996, 0), v100, z5, tool0;
MoveL Offs(p0,353.5,206.5, 0), v100, z5, tool0;
MoveL Offs(p0,351.42300000000006,209.95070000000004, 0), v100, z5, tool0;
MoveL Offs(p0,349.4120000000001,213.3096000000001, 0), v100, z5, tool0;
MoveL Offs(p0,347.49699999999996,216.52689999999998, 0), v100, z5, tool0;
MoveL Offs(p0,345.708,219.5528, 0), v100, z5, tool0;
MoveL Offs(p0,344.075,222.3375, 0), v100, z5, tool0;
MoveL Offs(p0,342.62800000000004,224.8312, 0), v100, z5, tool0;
MoveL Offs(p0,341.39700000000005,226.98409999999998, 0), v100, z5, tool0;
MoveL Offs(p0,340.412,228.7464, 0), v100, z5, tool0;
MoveL Offs(p0,339.70300000000003,230.0683, 0), v100, z5, tool0;
MoveL Offs(p0,339.3,230.9, 0), v100, z5, tool0;
MoveL Offs(p0,338.9229000000001,231.8016, 0), v100, z5, tool0;
MoveL Offs(p0,338.63520000000005,232.54480000000004, 0), v100, z5, tool0;
MoveL Offs(p0,338.44230000000005,233.15719999999996, 0), v100, z5, tool0;
MoveL Offs(p0,338.3496,233.66640000000007, 0), v100, z5, tool0;
MoveL Offs(p0,338.3625,234.1, 0), v100, z5, tool0;
MoveL Offs(p0,338.4864,234.48559999999998, 0), v100, z5, tool0;
MoveL Offs(p0,338.7267,234.8508, 0), v100, z5, tool0;
MoveL Offs(p0,339.08880000000005,235.2232, 0), v100, z5, tool0;
MoveL Offs(p0,339.57810000000006,235.6304, 0), v100, z5, tool0;
MoveL Offs(p0,340.2,236.1, 0), v100, z5, tool0;
MoveL Offs(p0,342.05740000000003,237.30630000000002, 0), v100, z5, tool0;
MoveL Offs(p0,344.06720000000007,238.2264000000001, 0), v100, z5, tool0;
MoveL Offs(p0,346.1958,238.86209999999997, 0), v100, z5, tool0;
MoveL Offs(p0,348.40960000000007,239.2152, 0), v100, z5, tool0;
MoveL Offs(p0,350.675,239.2875, 0), v100, z5, tool0;
MoveL Offs(p0,352.9584,239.0808, 0), v100, z5, tool0;
MoveL Offs(p0,355.22619999999995,238.5969, 0), v100, z5, tool0;
MoveL Offs(p0,357.44480000000004,237.8376, 0), v100, z5, tool0;
MoveL Offs(p0,359.5806,236.80470000000005, 0), v100, z5, tool0;
MoveL Offs(p0,361.6,235.5, 0), v100, z5, tool0;
MoveL Offs(p0,362.7103000000001,234.49080000000004, 0), v100, z5, tool0;
MoveL Offs(p0,363.87040000000013,233.16240000000002, 0), v100, z5, tool0;
MoveL Offs(p0,365.06409999999994,231.54359999999997, 0), v100, z5, tool0;
MoveL Offs(p0,366.27520000000004,229.66320000000002, 0), v100, z5, tool0;
MoveL Offs(p0,367.4875,227.55, 0), v100, z5, tool0;
MoveL Offs(p0,368.6848,225.2328, 0), v100, z5, tool0;
MoveL Offs(p0,369.8509,222.7404, 0), v100, z5, tool0;
MoveL Offs(p0,370.9696,220.10160000000002, 0), v100, z5, tool0;
MoveL Offs(p0,372.02470000000005,217.34520000000003, 0), v100, z5, tool0;
MoveL Offs(p0,373.0,214.5, 0), v100, z5, tool0;
MoveL Offs(p0,375.87430000000006,206.3605, 0), v100, z5, tool0;
MoveL Offs(p0,379.20640000000014,198.81200000000007, 0), v100, z5, tool0;
MoveL Offs(p0,382.9801,191.8695, 0), v100, z5, tool0;
MoveL Offs(p0,387.1792,185.54800000000003, 0), v100, z5, tool0;
MoveL Offs(p0,391.7875,179.8625, 0), v100, z5, tool0;
MoveL Offs(p0,396.7888,174.828, 0), v100, z5, tool0;
MoveL Offs(p0,402.1669,170.4595, 0), v100, z5, tool0;
MoveL Offs(p0,407.9056,166.77200000000002, 0), v100, z5, tool0;
MoveL Offs(p0,413.98870000000005,163.7805, 0), v100, z5, tool0;
MoveL Offs(p0,420.4,161.5, 0), v100, z5, tool0;
MoveL Offs(p0,423.15380000000005,160.848, 0), v100, z5, tool0;
MoveL Offs(p0,426.30240000000003,160.38800000000006, 0), v100, z5, tool0;
MoveL Offs(p0,429.7366,160.11399999999998, 0), v100, z5, tool0;
MoveL Offs(p0,433.3472,160.02, 0), v100, z5, tool0;
MoveL Offs(p0,437.025,160.1, 0), v100, z5, tool0;
MoveL Offs(p0,440.6608,160.348, 0), v100, z5, tool0;
MoveL Offs(p0,444.1454,160.75799999999998, 0), v100, z5, tool0;
MoveL Offs(p0,450.2242,162.04000000000002, 0), v100, z5, tool0;
MoveL Offs(p0,452.6,162.9, 0), v100, z5, tool0;
MoveL Offs(p0,454.4057000000001,163.78180000000003, 0), v100, z5, tool0;
MoveL Offs(p0,456.20960000000014,164.85440000000006, 0), v100, z5, tool0;
MoveL Offs(p0,457.9919,166.09859999999998, 0), v100, z5, tool0;
MoveL Offs(p0,459.73280000000005,167.4952, 0), v100, z5, tool0;
MoveL Offs(p0,461.4125,169.025, 0), v100, z5, tool0;
MoveL Offs(p0,463.01120000000003,170.6688, 0), v100, z5, tool0;
MoveL Offs(p0,464.50910000000005,172.4074, 0), v100, z5, tool0;
MoveL Offs(p0,465.88640000000004,174.22160000000002, 0), v100, z5, tool0;
MoveL Offs(p0,467.12330000000003,176.0922, 0), v100, z5, tool0;
MoveL Offs(p0,468.2,178.0, 0), v100, z5, tool0;
MoveL Offs(p0,469.11500000000007,180.1266, 0), v100, z5, tool0;
MoveL Offs(p0,469.82000000000016,182.50880000000006, 0), v100, z5, tool0;
MoveL Offs(p0,470.31499999999994,185.09019999999998, 0), v100, z5, tool0;
MoveL Offs(p0,470.6,187.8144, 0), v100, z5, tool0;
MoveL Offs(p0,470.675,190.625, 0), v100, z5, tool0;
MoveL Offs(p0,470.53999999999996,193.4656, 0), v100, z5, tool0;
MoveL Offs(p0,470.195,196.27979999999997, 0), v100, z5, tool0;
MoveL Offs(p0,469.64,199.0112, 0), v100, z5, tool0;
MoveL Offs(p0,468.875,201.60340000000002, 0), v100, z5, tool0;
MoveL Offs(p0,467.9,204.0, 0), v100, z5, tool0;
MoveL Offs(p0,466.00640000000004,207.5446, 0), v100, z5, tool0;
MoveL Offs(p0,463.7072000000001,210.96080000000006, 0), v100, z5, tool0;
MoveL Offs(p0,461.0347999999999,214.2222, 0), v100, z5, tool0;
MoveL Offs(p0,458.02160000000003,217.30239999999998, 0), v100, z5, tool0;
MoveL Offs(p0,454.7,220.175, 0), v100, z5, tool0;
MoveL Offs(p0,451.10240000000005,222.8136, 0), v100, z5, tool0;
MoveL Offs(p0,447.2611999999999,225.1918, 0), v100, z5, tool0;
MoveL Offs(p0,443.2088,227.28320000000002, 0), v100, z5, tool0;
MoveL Offs(p0,438.9776,229.0614, 0), v100, z5, tool0;
MoveL Offs(p0,434.6,230.5, 0), v100, z5, tool0;
MoveL Offs(p0,430.85810000000004,231.36510000000004, 0), v100, z5, tool0;
MoveL Offs(p0,426.8768000000001,231.8768000000001, 0), v100, z5, tool0;
MoveL Offs(p0,422.81270000000006,232.05970000000002, 0), v100, z5, tool0;
MoveL Offs(p0,418.82240000000013,231.9384, 0), v100, z5, tool0;
MoveL Offs(p0,415.0625,231.5375, 0), v100, z5, tool0;
MoveL Offs(p0,411.68960000000004,230.8816, 0), v100, z5, tool0;
MoveL Offs(p0,408.8603,229.9953, 0), v100, z5, tool0;
MoveL Offs(p0,406.73120000000006,228.90320000000003, 0), v100, z5, tool0;
MoveL Offs(p0,405.45889999999997,227.6299, 0), v100, z5, tool0;
MoveL Offs(p0,405.2,226.2, 0), v100, z5, tool0;
MoveL Offs(p0,405.7664000000002,225.31120000000004, 0), v100, z5, tool0;
MoveL Offs(p0,406.32409999999993,225.0093, 0), v100, z5, tool0;
MoveL Offs(p0,407.0912,224.8016, 0), v100, z5, tool0;
MoveL Offs(p0,408.0875,224.6875, 0), v100, z5, tool0;
MoveL Offs(p0,409.3328,224.6664, 0), v100, z5, tool0;
MoveL Offs(p0,410.8469,224.7377, 0), v100, z5, tool0;
MoveL Offs(p0,412.6496,224.90079999999998, 0), v100, z5, tool0;
MoveL Offs(p0,414.7607,225.15510000000003, 0), v100, z5, tool0;
MoveL Offs(p0,417.2,225.5, 0), v100, z5, tool0;
MoveL Offs(p0,419.91130000000004,225.7135, 0), v100, z5, tool0;
MoveL Offs(p0,425.9471,225.14450000000002, 0), v100, z5, tool0;
MoveL Offs(p0,429.15520000000004,224.404, 0), v100, z5, tool0;
MoveL Offs(p0,432.4125,223.3875, 0), v100, z5, tool0;
MoveL Offs(p0,435.6608,222.11599999999999, 0), v100, z5, tool0;
MoveL Offs(p0,438.8419,220.6105, 0), v100, z5, tool0;
MoveL Offs(p0,441.89760000000007,218.892, 0), v100, z5, tool0;
MoveL Offs(p0,444.7697,216.9815, 0), v100, z5, tool0;
MoveL Offs(p0,447.4,214.9, 0), v100, z5, tool0;
MoveL Offs(p0,448.99660000000006,213.3915, 0), v100, z5, tool0;
MoveL Offs(p0,450.53680000000014,211.76000000000008, 0), v100, z5, tool0;
MoveL Offs(p0,452.0062,210.0265, 0), v100, z5, tool0;
MoveL Offs(p0,453.39040000000006,208.21200000000005, 0), v100, z5, tool0;
MoveL Offs(p0,454.675,206.3375, 0), v100, z5, tool0;
MoveL Offs(p0,455.8456,204.424, 0), v100, z5, tool0;
MoveL Offs(p0,456.88779999999997,202.4925, 0), v100, z5, tool0;
MoveL Offs(p0,457.78720000000004,200.56400000000002, 0), v100, z5, tool0;
MoveL Offs(p0,458.5294,198.65950000000004, 0), v100, z5, tool0;
MoveL Offs(p0,459.1,196.8, 0), v100, z5, tool0;
MoveL Offs(p0,459.6938000000001,191.38440000000006, 0), v100, z5, tool0;
MoveL Offs(p0,458.6184000000001,186.42720000000006, 0), v100, z5, tool0;
MoveL Offs(p0,456.08859999999993,182.0328, 0), v100, z5, tool0;
MoveL Offs(p0,452.3192,178.3056, 0), v100, z5, tool0;
MoveL Offs(p0,447.525,175.35, 0), v100, z5, tool0;
MoveL Offs(p0,441.9208,173.27039999999997, 0), v100, z5, tool0;
MoveL Offs(p0,435.7214,172.1712, 0), v100, z5, tool0;
MoveL Offs(p0,429.14160000000004,172.15680000000003, 0), v100, z5, tool0;
MoveL Offs(p0,422.3962,173.3316, 0), v100, z5, tool0;
MoveL Offs(p0,415.7,175.8, 0), v100, z5, tool0;
MoveL Offs(p0,411.65170000000006,177.93920000000003, 0), v100, z5, tool0;
MoveL Offs(p0,407.88960000000014,180.48160000000007, 0), v100, z5, tool0;
MoveL Offs(p0,404.3879,183.4644, 0), v100, z5, tool0;
MoveL Offs(p0,401.12080000000003,186.9248, 0), v100, z5, tool0;
MoveL Offs(p0,398.0625,190.9, 0), v100, z5, tool0;
MoveL Offs(p0,395.18719999999996,195.42720000000003, 0), v100, z5, tool0;
MoveL Offs(p0,392.46909999999997,200.54360000000003, 0), v100, z5, tool0;
MoveL Offs(p0,389.8824000000001,206.28640000000001, 0), v100, z5, tool0;
MoveL Offs(p0,387.40130000000005,212.69279999999998, 0), v100, z5, tool0;
MoveL Offs(p0,385.0,219.8, 0), v100, z5, tool0;
MoveL Offs(p0,384.1632000000001,222.3376, 0), v100, z5, tool0;
MoveL Offs(p0,383.3336000000001,224.72880000000004, 0), v100, z5, tool0;
MoveL Offs(p0,382.51239999999996,226.97119999999995, 0), v100, z5, tool0;
MoveL Offs(p0,381.7008,229.06240000000003, 0), v100, z5, tool0;
MoveL Offs(p0,380.9,231.0, 0), v100, z5, tool0;
MoveL Offs(p0,380.1112,232.78159999999997, 0), v100, z5, tool0;
MoveL Offs(p0,379.3356,234.40479999999997, 0), v100, z5, tool0;
MoveL Offs(p0,378.5744,235.86720000000005, 0), v100, z5, tool0;
MoveL Offs(p0,377.8288,237.16639999999998, 0), v100, z5, tool0;
MoveL Offs(p0,377.1,238.3, 0), v100, z5, tool0;
MoveL Offs(p0,375.78120000000007,240.04620000000006, 0), v100, z5, tool0;
MoveL Offs(p0,374.3016000000001,241.73360000000008, 0), v100, z5, tool0;
MoveL Offs(p0,372.6864,243.34539999999998, 0), v100, z5, tool0;
MoveL Offs(p0,370.96079999999995,244.8648, 0), v100, z5, tool0;
MoveL Offs(p0,369.15,246.275, 0), v100, z5, tool0;
MoveL Offs(p0,367.2792,247.5592, 0), v100, z5, tool0;
MoveL Offs(p0,365.3736,248.70059999999998, 0), v100, z5, tool0;
MoveL Offs(p0,363.45840000000004,249.68240000000006, 0), v100, z5, tool0;
MoveL Offs(p0,361.5588,250.48780000000002, 0), v100, z5, tool0;
MoveL Offs(p0,359.7,251.1, 0), v100, z5, tool0;
MoveL Offs(p0,358.21470000000005,251.4125, 0), v100, z5, tool0;
MoveL Offs(p0,356.39760000000007,251.63200000000012, 0), v100, z5, tool0;
MoveL Offs(p0,354.3369,251.76149999999998, 0), v100, z5, tool0;
MoveL Offs(p0,352.12080000000003,251.804, 0), v100, z5, tool0;
MoveL Offs(p0,349.8375,251.7625, 0), v100, z5, tool0;
MoveL Offs(p0,347.5752,251.64000000000001, 0), v100, z5, tool0;
MoveL Offs(p0,345.42209999999994,251.4395, 0), v100, z5, tool0;
MoveL Offs(p0,341.79630000000003,250.8165, 0), v100, z5, tool0;
MoveL Offs(p0,340.5,250.4, 0), v100, z5, tool0;
MoveL Offs(p0,339.6312000000001,250.08080000000004, 0), v100, z5, tool0;
MoveL Offs(p0,339.34979999999996,250.0022, 0), v100, z5, tool0;
MoveL Offs(p0,339.16560000000004,249.9824, 0), v100, z5, tool0;
MoveL Offs(p0,339.075,250.025, 0), v100, z5, tool0;
MoveL Offs(p0,339.07439999999997,250.13360000000003, 0), v100, z5, tool0;
MoveL Offs(p0,339.5766,250.89140000000003, 0), v100, z5, tool0;
MoveL Offs(p0,339.9,251.3, 0), v100, z5, tool0;
MoveL Offs(p0,341.5987,252.68110000000007, 0), v100, z5, tool0;
MoveL Offs(p0,344.2976000000001,253.9848000000001, 0), v100, z5, tool0;
MoveL Offs(p0,347.8209,255.1817, 0), v100, z5, tool0;
MoveL Offs(p0,351.9928,256.24240000000003, 0), v100, z5, tool0;
MoveL Offs(p0,356.6375,257.1375, 0), v100, z5, tool0;
MoveL Offs(p0,361.5792,257.8376, 0), v100, z5, tool0;
MoveL Offs(p0,366.64209999999997,258.3133, 0), v100, z5, tool0;
MoveL Offs(p0,371.65040000000005,258.53520000000003, 0), v100, z5, tool0;
MoveL Offs(p0,376.4283,258.4739, 0), v100, z5, tool0;
MoveL Offs(p0,380.8,258.1, 0), v100, z5, tool0;
MoveL Offs(p0,384.1562,257.69680000000005, 0), v100, z5, tool0;
MoveL Offs(p0,386.9016000000001,257.3944000000001, 0), v100, z5, tool0;
MoveL Offs(p0,389.1214,257.2036, 0), v100, z5, tool0;
MoveL Offs(p0,390.90080000000006,257.13520000000005, 0), v100, z5, tool0;
MoveL Offs(p0,392.325,257.2, 0), v100, z5, tool0;
MoveL Offs(p0,393.4792,257.4088, 0), v100, z5, tool0;
MoveL Offs(p0,394.4486,257.7724, 0), v100, z5, tool0;
MoveL Offs(p0,395.3184,258.30160000000006, 0), v100, z5, tool0;
MoveL Offs(p0,396.1738,259.0072, 0), v100, z5, tool0;
MoveL Offs(p0,397.1,259.9, 0), v100, z5, tool0;
MoveL Offs(p0,398.3268000000001,261.27320000000003, 0), v100, z5, tool0;
MoveL Offs(p0,399.2464000000001,262.64160000000004, 0), v100, z5, tool0;
MoveL Offs(p0,399.8576,264.0184, 0), v100, z5, tool0;
MoveL Offs(p0,400.1592,265.4168, 0), v100, z5, tool0;
MoveL Offs(p0,400.15,266.85, 0), v100, z5, tool0;
MoveL Offs(p0,399.82879999999994,268.33119999999997, 0), v100, z5, tool0;
MoveL Offs(p0,399.19440000000003,269.8736, 0), v100, z5, tool0;
MoveL Offs(p0,398.2456,271.4904, 0), v100, z5, tool0;
MoveL Offs(p0,395.4,275.0, 0), v100, z5, tool0;
MoveL Offs(p0,393.70420000000007,276.93120000000005, 0), v100, z5, tool0;
MoveL Offs(p0,392.3336000000001,278.78560000000004, 0), v100, z5, tool0;
MoveL Offs(p0,391.28340000000003,280.5944, 0), v100, z5, tool0;
MoveL Offs(p0,390.5488000000001,282.3888, 0), v100, z5, tool0;
MoveL Offs(p0,390.125,284.2, 0), v100, z5, tool0;
MoveL Offs(p0,390.0072,286.05920000000003, 0), v100, z5, tool0;
MoveL Offs(p0,390.1906,287.99760000000003, 0), v100, z5, tool0;
MoveL Offs(p0,390.6704000000001,290.04640000000006, 0), v100, z5, tool0;
MoveL Offs(p0,391.4418,292.2368, 0), v100, z5, tool0;
MoveL Offs(p0,392.5,294.6, 0), v100, z5, tool0;
MoveL Offs(p0,393.4861,296.4208, 0), v100, z5, tool0;
MoveL Offs(p0,394.5568000000001,298.0664000000001, 0), v100, z5, tool0;
MoveL Offs(p0,395.76070000000004,299.5716, 0), v100, z5, tool0;
MoveL Offs(p0,397.1464000000001,300.9712, 0), v100, z5, tool0;
MoveL Offs(p0,398.7625,302.3, 0), v100, z5, tool0;
MoveL Offs(p0,400.6576,303.5928, 0), v100, z5, tool0;
MoveL Offs(p0,402.8803,304.8844, 0), v100, z5, tool0;
MoveL Offs(p0,405.47920000000005,306.2096, 0), v100, z5, tool0;
MoveL Offs(p0,408.50290000000007,307.6032, 0), v100, z5, tool0;
MoveL Offs(p0,412.0,309.1, 0), v100, z5, tool0;
MoveL Offs(p0,413.3224,309.65920000000006, 0), v100, z5, tool0;
MoveL Offs(p0,414.63520000000005,310.2496000000001, 0), v100, z5, tool0;
MoveL Offs(p0,415.91679999999997,310.86039999999997, 0), v100, z5, tool0;
MoveL Offs(p0,417.1456,311.48080000000004, 0), v100, z5, tool0;
MoveL Offs(p0,418.3,312.1, 0), v100, z5, tool0;
MoveL Offs(p0,419.35839999999996,312.70719999999994, 0), v100, z5, tool0;
MoveL Offs(p0,420.29920000000004,313.2916, 0), v100, z5, tool0;
MoveL Offs(p0,421.10080000000005,313.84240000000005, 0), v100, z5, tool0;
MoveL Offs(p0,421.7416,314.34880000000004, 0), v100, z5, tool0;
MoveL Offs(p0,422.2,314.8, 0), v100, z5, tool0;
MoveL Offs(p0,423.1301,315.9451, 0), v100, z5, tool0;
MoveL Offs(p0,423.82080000000013,317.21680000000003, 0), v100, z5, tool0;
MoveL Offs(p0,424.2727,318.6097, 0), v100, z5, tool0;
MoveL Offs(p0,424.48640000000006,320.1184, 0), v100, z5, tool0;
MoveL Offs(p0,424.4625,321.7375, 0), v100, z5, tool0;
MoveL Offs(p0,424.20160000000004,323.4616, 0), v100, z5, tool0;
MoveL Offs(p0,423.7043,325.2853, 0), v100, z5, tool0;
MoveL Offs(p0,422.97120000000007,327.20320000000004, 0), v100, z5, tool0;
MoveL Offs(p0,420.8,331.3, 0), v100, z5, tool0;
MoveL Offs(p0,419.46060000000006,333.57120000000003, 0), v100, z5, tool0;
MoveL Offs(p0,418.31680000000017,335.78960000000006, 0), v100, z5, tool0;
MoveL Offs(p0,417.36019999999996,337.9924, 0), v100, z5, tool0;
MoveL Offs(p0,416.58240000000006,340.21680000000003, 0), v100, z5, tool0;
MoveL Offs(p0,415.975,342.5, 0), v100, z5, tool0;
MoveL Offs(p0,415.5296,344.87919999999997, 0), v100, z5, tool0;
MoveL Offs(p0,415.2378,347.3916, 0), v100, z5, tool0;
MoveL Offs(p0,415.0912,350.0744, 0), v100, z5, tool0;
MoveL Offs(p0,415.08140000000003,352.9648, 0), v100, z5, tool0;
MoveL Offs(p0,415.2,356.1, 0), v100, z5, tool0;
MoveL Offs(p0,415.5077,359.57720000000006, 0), v100, z5, tool0;
MoveL Offs(p0,416.00560000000013,362.8576000000001, 0), v100, z5, tool0;
MoveL Offs(p0,416.68590000000006,365.9244, 0), v100, z5, tool0;
MoveL Offs(p0,417.54080000000005,368.7608, 0), v100, z5, tool0;
MoveL Offs(p0,418.5625,371.35, 0), v100, z5, tool0;
MoveL Offs(p0,419.7432,373.67519999999996, 0), v100, z5, tool0;
MoveL Offs(p0,421.0751,375.7196, 0), v100, z5, tool0;
MoveL Offs(p0,422.5504000000001,377.4664, 0), v100, z5, tool0;
MoveL Offs(p0,424.16130000000004,378.89880000000005, 0), v100, z5, tool0;
MoveL Offs(p0,425.9,380.0, 0), v100, z5, tool0;
MoveL Offs(p0,427.1838000000001,380.7166, 0), v100, z5, tool0;
MoveL Offs(p0,428.27440000000007,381.48480000000006, 0), v100, z5, tool0;
MoveL Offs(p0,429.17060000000004,382.30219999999997, 0), v100, z5, tool0;
MoveL Offs(p0,429.87120000000004,383.16640000000007, 0), v100, z5, tool0;
MoveL Offs(p0,430.375,384.075, 0), v100, z5, tool0;
MoveL Offs(p0,430.6808,385.0256, 0), v100, z5, tool0;
MoveL Offs(p0,430.7874,386.0158, 0), v100, z5, tool0;
MoveL Offs(p0,430.69360000000006,387.0432, 0), v100, z5, tool0;
MoveL Offs(p0,430.3982,388.10540000000003, 0), v100, z5, tool0;
MoveL Offs(p0,429.9,389.2, 0), v100, z5, tool0;
MoveL Offs(p0,429.454,390.03540000000004, 0), v100, z5, tool0;
MoveL Offs(p0,429.00800000000015,390.74720000000013, 0), v100, z5, tool0;
MoveL Offs(p0,428.55,391.3438, 0), v100, z5, tool0;
MoveL Offs(p0,428.06800000000004,391.83360000000005, 0), v100, z5, tool0;
MoveL Offs(p0,427.55,392.225, 0), v100, z5, tool0;
MoveL Offs(p0,426.9839999999999,392.52639999999997, 0), v100, z5, tool0;
MoveL Offs(p0,426.358,392.7462, 0), v100, z5, tool0;
MoveL Offs(p0,425.66,392.8928000000001, 0), v100, z5, tool0;
MoveL Offs(p0,424.87800000000004,392.9746, 0), v100, z5, tool0;
MoveL Offs(p0,424.0,393.0, 0), v100, z5, tool0;
MoveL Offs(p0,421.8991000000001,392.48420000000004, 0), v100, z5, tool0;
MoveL Offs(p0,418.62880000000007,390.9976000000001, 0), v100, z5, tool0;
MoveL Offs(p0,414.32769999999994,388.6314, 0), v100, z5, tool0;
MoveL Offs(p0,409.1344,385.4768, 0), v100, z5, tool0;
MoveL Offs(p0,403.1875,381.625, 0), v100, z5, tool0;
MoveL Offs(p0,396.62559999999996,377.1672, 0), v100, z5, tool0;
MoveL Offs(p0,389.5873,372.1946, 0), v100, z5, tool0;
MoveL Offs(p0,382.2112,366.7984, 0), v100, z5, tool0;
MoveL Offs(p0,374.6359,361.06980000000004, 0), v100, z5, tool0;
MoveL Offs(p0,367.0,355.1, 0), v100, z5, tool0;
MoveL Offs(p0,354.5,345.2, 0), v100, z5, tool0;
MoveL Offs(p0,353.7,348.2, 0), v100, z5, tool0;
MoveL Offs(p0,353.0339,350.31230000000005, 0), v100, z5, tool0;
MoveL Offs(p0,352.2352000000001,352.0904000000001, 0), v100, z5, tool0;
MoveL Offs(p0,351.30330000000004,353.5361, 0), v100, z5, tool0;
MoveL Offs(p0,350.23760000000004,354.6512000000001, 0), v100, z5, tool0;
MoveL Offs(p0,349.0375,355.4375, 0), v100, z5, tool0;
MoveL Offs(p0,347.7024,355.8968, 0), v100, z5, tool0;
MoveL Offs(p0,346.2317,356.03090000000003, 0), v100, z5, tool0;
MoveL Offs(p0,344.62480000000005,355.8416, 0), v100, z5, tool0;
MoveL Offs(p0,342.8811,355.3307, 0), v100, z5, tool0;
MoveL Offs(p0,341.0,354.5, 0), v100, z5, tool0;
MoveL Offs(p0,340.35710000000006,354.17300000000006, 0), v100, z5, tool0;
MoveL Offs(p0,339.8048000000001,353.9120000000001, 0), v100, z5, tool0;
MoveL Offs(p0,339.3377,353.717, 0), v100, z5, tool0;
MoveL Offs(p0,338.95040000000006,353.588, 0), v100, z5, tool0;
MoveL Offs(p0,338.6375,353.525, 0), v100, z5, tool0;
MoveL Offs(p0,338.3936,353.52799999999996, 0), v100, z5, tool0;
MoveL Offs(p0,338.2133,353.59700000000004, 0), v100, z5, tool0;
MoveL Offs(p0,338.0912,353.732, 0), v100, z5, tool0;
MoveL Offs(p0,338.0219,353.933, 0), v100, z5, tool0;
MoveL Offs(p0,338.0,354.2, 0), v100, z5, tool0;
MoveL Offs(p0,337.76000000000005,356.3824000000001, 0), v100, z5, tool0;
MoveL Offs(p0,337.48699999999997,357.5561, 0), v100, z5, tool0;
MoveL Offs(p0,337.136,358.7232, 0), v100, z5, tool0;
MoveL Offs(p0,336.725,359.8375, 0), v100, z5, tool0;
MoveL Offs(p0,336.27199999999993,360.8528, 0), v100, z5, tool0;
MoveL Offs(p0,335.79499999999996,361.72290000000004, 0), v100, z5, tool0;
MoveL Offs(p0,335.312,362.40160000000003, 0), v100, z5, tool0;
MoveL Offs(p0,334.841,362.84270000000004, 0), v100, z5, tool0;
MoveL Offs(p0,334.4,363.0, 0), v100, z5, tool0;
MoveL Offs(p0,333.25200000000007,362.7392000000001, 0), v100, z5, tool0;
MoveL Offs(p0,332.22200000000004,362.43029999999993, 0), v100, z5, tool0;
MoveL Offs(p0,330.928,362.01759999999996, 0), v100, z5, tool0;
MoveL Offs(p0,329.4,361.5125, 0), v100, z5, tool0;
MoveL Offs(p0,327.668,360.9264, 0), v100, z5, tool0;
MoveL Offs(p0,325.762,360.27070000000003, 0), v100, z5, tool0;
MoveL Offs(p0,323.71200000000005,359.5568, 0), v100, z5, tool0;
MoveL Offs(p0,321.548,358.7961, 0), v100, z5, tool0;
MoveL Offs(p0,319.3,358.0, 0), v100, z5, tool0;
MoveL Offs(p0,317.0938,357.1825, 0), v100, z5, tool0;
MoveL Offs(p0,314.9944000000001,356.41600000000005, 0), v100, z5, tool0;
MoveL Offs(p0,313.0306,355.7095, 0), v100, z5, tool0;
MoveL Offs(p0,311.23120000000006,355.07200000000006, 0), v100, z5, tool0;
MoveL Offs(p0,309.625,354.5125, 0), v100, z5, tool0;
MoveL Offs(p0,308.24080000000004,354.03999999999996, 0), v100, z5, tool0;
MoveL Offs(p0,307.1074,353.6635, 0), v100, z5, tool0;
MoveL Offs(p0,306.2536,353.392, 0), v100, z5, tool0;
MoveL Offs(p0,305.70820000000003,353.2345, 0), v100, z5, tool0;
MoveL Offs(p0,305.5,353.2, 0), v100, z5, tool0;
MoveL Offs(p0,305.8624000000001,354.1040000000001, 0), v100, z5, tool0;
MoveL Offs(p0,306.33610000000004,355.0945, 0), v100, z5, tool0;
MoveL Offs(p0,306.9832,356.4, 0), v100, z5, tool0;
MoveL Offs(p0,307.7875,357.9875, 0), v100, z5, tool0;
MoveL Offs(p0,308.73279999999994,359.82399999999996, 0), v100, z5, tool0;
MoveL Offs(p0,309.8029,361.8765, 0), v100, z5, tool0;
MoveL Offs(p0,310.98159999999996,364.11199999999997, 0), v100, z5, tool0;
MoveL Offs(p0,312.2527,366.4975, 0), v100, z5, tool0;
MoveL Offs(p0,313.6,369.0, 0), v100, z5, tool0;
MoveL Offs(p0,315.3148,372.2107, 0), v100, z5, tool0;
MoveL Offs(p0,316.8064000000001,375.0776000000001, 0), v100, z5, tool0;
MoveL Offs(p0,318.0856,377.62289999999996, 0), v100, z5, tool0;
MoveL Offs(p0,319.1632,379.8688000000001, 0), v100, z5, tool0;
MoveL Offs(p0,320.05,381.8375, 0), v100, z5, tool0;
MoveL Offs(p0,320.7568,383.5512, 0), v100, z5, tool0;
MoveL Offs(p0,321.29439999999994,385.0321, 0), v100, z5, tool0;
MoveL Offs(p0,321.67359999999996,386.30240000000003, 0), v100, z5, tool0;
MoveL Offs(p0,321.9052,387.3843, 0), v100, z5, tool0;
MoveL Offs(p0,322.0,388.3, 0), v100, z5, tool0;
MoveL Offs(p0,321.4488000000001,391.5984000000001, 0), v100, z5, tool0;
MoveL Offs(p0,320.8012,392.9476, 0), v100, z5, tool0;
MoveL Offs(p0,319.9424,394.07120000000003, 0), v100, z5, tool0;
MoveL Offs(p0,318.9,394.95, 0), v100, z5, tool0;
MoveL Offs(p0,317.7016,395.5648, 0), v100, z5, tool0;
MoveL Offs(p0,316.37479999999994,395.89639999999997, 0), v100, z5, tool0;
MoveL Offs(p0,314.9472,395.92560000000003, 0), v100, z5, tool0;
MoveL Offs(p0,313.4464,395.6332, 0), v100, z5, tool0;
MoveL Offs(p0,311.9,395.0, 0), v100, z5, tool0;
MoveL Offs(p0,311.47810000000004,394.6568, 0), v100, z5, tool0;
MoveL Offs(p0,310.8288000000001,394.0064000000001, 0), v100, z5, tool0;
MoveL Offs(p0,309.9767,393.07759999999996, 0), v100, z5, tool0;
MoveL Offs(p0,308.9464,391.8992, 0), v100, z5, tool0;
MoveL Offs(p0,307.7625,390.5, 0), v100, z5, tool0;
MoveL Offs(p0,306.44960000000003,388.9088, 0), v100, z5, tool0;
MoveL Offs(p0,305.03229999999996,387.1544, 0), v100, z5, tool0;
MoveL Offs(p0,303.53520000000003,385.2656, 0), v100, z5, tool0;
MoveL Offs(p0,301.9829,383.2712, 0), v100, z5, tool0;
MoveL Offs(p0,300.4,381.2, 0), v100, z5, tool0;
MoveL Offs(p0,298.0783,378.11930000000007, 0), v100, z5, tool0;
MoveL Offs(p0,296.1184000000001,375.56240000000014, 0), v100, z5, tool0;
